LIN {X 0,Y 339.349,Z 929.895,A -85,B 0,C 180,E1 -14128.813,E2 -14128.813} C_VEL
LIN {X 0,Y 339.347,Z 930.371,A -85,B 0,C 180,E1 -14130,E2 -14130} C_VEL
LIN {X 0,Y 339.321,Z 930.387,A -85,B 0,C 180,E1 -14131.187,E2 -14131.187} C_VEL
LIN {X 0,Y 339.177,Z 929.963,A -85,B 0,C 180,E1 -14132.375,E2 -14132.375} C_VEL
LIN {X 0,Y 339.147,Z 929.133,A -85,B 0,C 180,E1 -14133.564,E2 -14133.564} C_VEL
LIN {X 0,Y 339.18,Z 927.893,A -85,B 0,C 180,E1 -14134.754,E2 -14134.754} C_VEL
LIN {X 0,Y 339.253,Z 925.189,A -85,B 0,C 180,E1 -14136.542,E2 -14136.542} C_VEL
LIN {X 0,Y 339.515,Z 921.472,A -85,B 0,C 180,E1 -14138.332,E2 -14138.332} C_VEL
LIN {X 0,Y 339.961,Z 916.67,A -85,B 0,C 180,E1 -14140.121,E2 -14140.121} C_VEL
LIN {X 0,Y 340.849,Z 909.521,A -85,B 0,C 180,E1 -14142.201,E2 -14142.201} C_VEL
LIN {X 0,Y 341.955,Z 901.959,A -85,B 0,C 180,E1 -14143.975,E2 -14143.975} C_VEL
LIN {X 0,Y 343.322,Z 892.798,A -85,B 0,C 180,E1 -14145.731,E2 -14145.731} C_VEL
LIN {X 0,Y 344.863,Z 882.415,A -85,B 0,C 180,E1 -14147.34,E2 -14147.34} C_VEL
LIN {X 0,Y 346.714,Z 871.123,A -85,B 0,C 180,E1 -14148.771,E2 -14148.771} C_VEL
LIN {X 0,Y 347.214,Z 865.96,A -85,B 0,C 180,E1 -14149.357,E2 -14149.357} C_VEL
LIN {X 0,Y 347.253,Z 853.333,A -85,B 0,C 180,E1 -14150.673,E2 -14150.673} C_VEL
LIN {X 0,Y 346.425,Z 843.606,A -85,B 0,C 180,E1 -14151.619,E2 -14151.619} C_VEL
LIN {X 0,Y 344.27,Z 832.038,A -85,B 0,C 180,E1 -14152.71,E2 -14152.71} C_VEL
LIN {X 0,Y 341.467,Z 821.968,A -85,B 0,C 180,E1 -14153.676,E2 -14153.676} C_VEL
LIN {X 0,Y 340.675,Z 818.661,A -85,B 0,C 180,E1 -14153.963,E2 -14153.963} C_VEL
LIN {X 0,Y 341.252,Z 813.344,A -85,B 0,C 180,E1 -14156.942,E2 -14156.942} C_VEL
LIN {X 0,Y 342.064,Z 807.69,A -85,B 0,C 180,E1 -14160.352,E2 -14160.352} C_VEL
LIN {X 0,Y 343.055,Z 802.834,A -85,B 0,C 180,E1 -14163.583,E2 -14163.583} C_VEL
LIN {X 0,Y 343.614,Z 799.164,A -85,B 0,C 180,E1 -14166.381,E2 -14166.381} C_VEL
LIN {X 0,Y 343.643,Z 796.286,A -85,B 0,C 180,E1 -14168.998,E2 -14168.998} C_VEL
LIN {X 0,Y 343.254,Z 793.267,A -85,B 0,C 180,E1 -14172.515,E2 -14172.515} C_VEL
LIN {X 0,Y 342.871,Z 791.214,A -85,B 0,C 180,E1 -14175.841,E2 -14175.841} C_VEL
LIN {X 0,Y 342.57,Z 789.841,A -85,B 0,C 180,E1 -14179.383,E2 -14179.383} C_VEL
LIN {X 0,Y 342.384,Z 789.323,A -85,B 0,C 180,E1 -14181.989,E2 -14181.989} C_VEL
LIN {X 0,Y 342.116,Z 789.226,A -85,B 0,C 180,E1 -14185.257,E2 -14185.257} C_VEL
LIN {X 0,Y 341.816,Z 789.514,A -85,B 0,C 180,E1 -14187.683,E2 -14187.683} C_VEL
LIN {X 0,Y 341.448,Z 790.146,A -85,B 0,C 180,E1 -14190.396,E2 -14190.396} C_VEL
LIN {X 0,Y 341.157,Z 791.012,A -85,B 0,C 180,E1 -14193.049,E2 -14193.049} C_VEL
LIN {X 0,Y 340.825,Z 792.487,A -85,B 0,C 180,E1 -14196.25,E2 -14196.25} C_VEL
LIN {X 0,Y 341.966,Z 795.393,A -85,B 0,C 180,E1 -14196.585,E2 -14196.585} C_VEL
LIN {X 0,Y 345.202,Z 802.217,A -85,B 0,C 180,E1 -14197.481,E2 -14197.481} C_VEL
LIN {X 0,Y 348.415,Z 810.639,A -85,B 0,C 180,E1 -14198.542,E2 -14198.542} C_VEL
LIN {X 0,Y 350.867,Z 820.747,A -85,B 0,C 180,E1 -14199.771,E2 -14199.771} C_VEL
LIN {X 0,Y 349.277,Z 832.605,A -85,B 0,C 180,E1 -14200.944,E2 -14200.944} C_VEL
LIN {X 0,Y 347.586,Z 843.821,A -85,B 0,C 180,E1 -14202.343,E2 -14202.343} C_VEL
LIN {X 0,Y 345.99,Z 853.23,A -85,B 0,C 180,E1 -14203.78,E2 -14203.78} C_VEL
LIN {X 0,Y 344.569,Z 861.071,A -85,B 0,C 180,E1 -14205.228,E2 -14205.228} C_VEL
LIN {X 0,Y 343.208,Z 868.826,A -85,B 0,C 180,E1 -14206.981,E2 -14206.981} C_VEL
LIN {X 0,Y 342.084,Z 875.111,A -85,B 0,C 180,E1 -14208.744,E2 -14208.744} C_VEL
LIN {X 0,Y 341.237,Z 880.125,A -85,B 0,C 180,E1 -14210.515,E2 -14210.515} C_VEL
LIN {X 0,Y 340.659,Z 883.491,A -85,B 0,C 180,E1 -14212.002,E2 -14212.002} C_VEL
LIN {X 0,Y 339.84,Z 886.98,A -85,B 0,C 180,E1 -14214.064,E2 -14214.064} C_VEL
LIN {X 0,Y 339.857,Z 888.363,A -85,B 0,C 180,E1 -14215.254,E2 -14215.254} C_VEL
LIN {X 0,Y 339.695,Z 889.321,A -85,B 0,C 180,E1 -14216.44,E2 -14216.44} C_VEL
LIN {X 0,Y 339.399,Z 890.044,A -85,B 0,C 180,E1 -14218.812,E2 -14218.812} C_VEL
LIN {X 0,Y 339.348,Z 889.81,A -85,B 0,C 180,E1 -14219.999,E2 -14219.999} C_VEL
LIN {X 0,Y 339.359,Z 889.126,A -85,B 0,C 180,E1 -14221.185,E2 -14221.185} C_VEL
LIN {X 0,Y 339.359,Z 888.038,A -85,B 0,C 180,E1 -14222.373,E2 -14222.373} C_VEL
LIN {X 0,Y 339.34,Z 886.549,A -85,B 0,C 180,E1 -14223.561,E2 -14223.561} C_VEL
LIN {X 0,Y 339.555,Z 883.457,A -85,B 0,C 180,E1 -14225.343,E2 -14225.343} C_VEL
LIN {X 0,Y 339.828,Z 879.306,A -85,B 0,C 180,E1 -14227.127,E2 -14227.127} C_VEL
LIN {X 0,Y 340.296,Z 872.949,A -85,B 0,C 180,E1 -14229.209,E2 -14229.209} C_VEL
LIN {X 0,Y 340.943,Z 866.043,A -85,B 0,C 180,E1 -14230.991,E2 -14230.991} C_VEL
LIN {X 0,Y 341.715,Z 857.519,A -85,B 0,C 180,E1 -14232.772,E2 -14232.772} C_VEL
LIN {X 0,Y 342.637,Z 848.818,A -85,B 0,C 180,E1 -14234.248,E2 -14234.248} C_VEL
LIN {X 0,Y 343.617,Z 838.67,A -85,B 0,C 180,E1 -14235.667,E2 -14235.667} C_VEL
LIN {X 0,Y 344.465,Z 827.918,A -85,B 0,C 180,E1 -14236.901,E2 -14236.901} C_VEL
LIN {X 0,Y 345.434,Z 815.586,A -85,B 0,C 180,E1 -14238.022,E2 -14238.022} C_VEL
LIN {X 0,Y 345.337,Z 812.445,A -85,B 0,C 180,E1 -14238.283,E2 -14238.283} C_VEL
LIN {X 0,Y 342.494,Z 799.34,A -85,B 0,C 180,E1 -14239.278,E2 -14239.278} C_VEL
LIN {X 0,Y 339.507,Z 785.356,A -85,B 0,C 180,E1 -14240.088,E2 -14240.088} C_VEL
LIN {X 0,Y 339.632,Z 781.305,A -85,B 0,C 180,E1 -14244.446,E2 -14244.446} C_VEL
LIN {X 0,Y 339.737,Z 779.169,A -85,B 0,C 180,E1 -14247.186,E2 -14247.186} C_VEL
LIN {X 0,Y 340.169,Z 779.109,A -85,B 0,C 180,E1 -14251.097,E2 -14251.097} C_VEL
LIN {X 0,Y 340.534,Z 779.069,A -85,B 0,C 180,E1 -14254.358,E2 -14254.358} C_VEL
LIN {X 0,Y 340.668,Z 779.051,A -85,B 0,C 180,E1 -14256.744,E2 -14256.744} C_VEL
LIN {X 0,Y 340.694,Z 779.044,A -85,B 0,C 180,E1 -14259.751,E2 -14259.751} C_VEL
LIN {X 0,Y 340.671,Z 779.05,A -85,B 0,C 180,E1 -14262.903,E2 -14262.903} C_VEL
LIN {X 0,Y 340.67,Z 779.05,A -85,B 0,C 180,E1 -14267.095,E2 -14267.095} C_VEL
LIN {X 0,Y 340.692,Z 779.044,A -85,B 0,C 180,E1 -14270.246,E2 -14270.246} C_VEL
LIN {X 0,Y 340.703,Z 779.043,A -85,B 0,C 180,E1 -14273.558,E2 -14273.558} C_VEL
LIN {X 0,Y 340.685,Z 779.044,A -85,B 0,C 180,E1 -14276.152,E2 -14276.152} C_VEL
LIN {X 0,Y 340.716,Z 779.041,A -85,B 0,C 180,E1 -14280.033,E2 -14280.033} C_VEL
LIN {X 0,Y 340.715,Z 779.044,A -85,B 0,C 180,E1 -14283.012,E2 -14283.012} C_VEL
LIN {X 0,Y 340.734,Z 779.041,A -85,B 0,C 180,E1 -14285.637,E2 -14285.637} C_VEL
LIN {X 0,Y 340.722,Z 779.046,A -85,B 0,C 180,E1 -14289.472,E2 -14289.472} C_VEL
LIN {X 0,Y 340.783,Z 779.034,A -85,B 0,C 180,E1 -14291.98,E2 -14291.98} C_VEL
LIN {X 0,Y 340.861,Z 779.028,A -85,B 0,C 180,E1 -14295.705,E2 -14295.705} C_VEL
LIN {X 0,Y 340.838,Z 779.028,A -85,B 0,C 180,E1 -14299.305,E2 -14299.305} C_VEL
LIN {X 0,Y 340.99,Z 779.006,A -85,B 0,C 180,E1 -14302.896,E2 -14302.896} C_VEL
LIN {X 0,Y 340.798,Z 779.031,A -85,B 0,C 180,E1 -14305.268,E2 -14305.268} C_VEL
LIN {X 0,Y 341.114,Z 778.994,A -85,B 0,C 180,E1 -14307.638,E2 -14307.638} C_VEL
LIN {X 0,Y 341.077,Z 778.995,A -85,B 0,C 180,E1 -14311.181,E2 -14311.181} C_VEL
LIN {X 0,Y 341.106,Z 778.995,A -85,B 0,C 180,E1 -14312.362,E2 -14312.362} C_VEL
LIN {X 0,Y 341.001,Z 779.008,A -85,B 0,C 180,E1 -14315.915,E2 -14315.915} C_VEL
LIN {X 0,Y 340.954,Z 779.016,A -85,B 0,C 180,E1 -14318.356,E2 -14318.356} C_VEL
LIN {X 0,Y 340.835,Z 779.028,A -85,B 0,C 180,E1 -14321.9,E2 -14321.9} C_VEL
LIN {X 0,Y 340.808,Z 779.029,A -85,B 0,C 180,E1 -14325.55,E2 -14325.55} C_VEL
LIN {X 0,Y 340.726,Z 779.039,A -85,B 0,C 180,E1 -14329.27,E2 -14329.27} C_VEL
LIN {X 0,Y 340.705,Z 779.044,A -85,B 0,C 180,E1 -14333.075,E2 -14333.075} C_VEL
LIN {X 0,Y 340.712,Z 779.041,A -85,B 0,C 180,E1 -14335.669,E2 -14335.669} C_VEL
LIN {X 0,Y 340.7,Z 779.043,A -85,B 0,C 180,E1 -14339.675,E2 -14339.675} C_VEL
LIN {X 0,Y 340.679,Z 779.047,A -85,B 0,C 180,E1 -14342.437,E2 -14342.437} C_VEL
LIN {X 0,Y 340.711,Z 779.044,A -85,B 0,C 180,E1 -14345.28,E2 -14345.28} C_VEL
LIN {X 0,Y 340.703,Z 779.043,A -85,B 0,C 180,E1 -14348.387,E2 -14348.387} C_VEL
LIN {X 0,Y 340.693,Z 779.044,A -85,B 0,C 180,E1 -14352.047,E2 -14352.047} C_VEL
LIN {X 0,Y 340.647,Z 779.049,A -85,B 0,C 180,E1 -14356.228,E2 -14356.228} C_VEL
LIN {X 0,Y 340.684,Z 779.047,A -85,B 0,C 180,E1 -14359.754,E2 -14359.754} C_VEL
LIN {X 0,Y 340.722,Z 779.043,A -85,B 0,C 180,E1 -14361.773,E2 -14361.773} C_VEL
LIN {X 0,Y 340.599,Z 779.055,A -85,B 0,C 180,E1 -14364.709,E2 -14364.709} C_VEL
LIN {X 0,Y 340.366,Z 779.088,A -85,B 0,C 180,E1 -14367.842,E2 -14367.842} C_VEL
LIN {X 0,Y 339.991,Z 779.131,A -85,B 0,C 180,E1 -14370.681,E2 -14370.681} C_VEL
LIN {X 0,Y 339.185,Z 779.237,A -85,B 0,C 180,E1 -14371.668,E2 -14371.668} C_VEL
LIN {X 0,Y 336.112,Z 779.617,A -85,B 0,C 180,E1 -14373.268,E2 -14373.268} C_VEL
LIN {X 0,Y 333.564,Z 780.155,A -85,B 0,C 180,E1 -14374.56,E2 -14374.56} C_VEL
LIN {X 0,Y 332.467,Z 780.857,A -85,B 0,C 180,E1 -14375.557,E2 -14375.557} C_VEL
LIN {X 0,Y 332.373,Z 781.177,A -85,B 0,C 180,E1 -14375.893,E2 -14375.893} C_VEL
LIN {X 0,Y 332.385,Z 785.144,A -85,B 0,C 180,E1 -14379.744,E2 -14379.744} C_VEL
LIN {X 0,Y 335.629,Z 800.339,A -85,B 0,C 180,E1 -14380.665,E2 -14380.665} C_VEL
LIN {X 0,Y 338.393,Z 814.066,A -85,B 0,C 180,E1 -14381.752,E2 -14381.752} C_VEL
LIN {X 0,Y 337.495,Z 826.677,A -85,B 0,C 180,E1 -14382.895,E2 -14382.895} C_VEL
LIN {X 0,Y 336.561,Z 838.501,A -85,B 0,C 180,E1 -14384.25,E2 -14384.25} C_VEL
LIN {X 0,Y 335.519,Z 849.022,A -85,B 0,C 180,E1 -14385.753,E2 -14385.753} C_VEL
LIN {X 0,Y 334.627,Z 857.724,A -85,B 0,C 180,E1 -14387.261,E2 -14387.261} C_VEL
LIN {X 0,Y 333.809,Z 866.28,A -85,B 0,C 180,E1 -14389.079,E2 -14389.079} C_VEL
LIN {X 0,Y 333.128,Z 873.174,A -85,B 0,C 180,E1 -14390.897,E2 -14390.897} C_VEL
LIN {X 0,Y 332.756,Z 878.716,A -85,B 0,C 180,E1 -14392.721,E2 -14392.721} C_VEL
LIN {X 0,Y 332.459,Z 883.055,A -85,B 0,C 180,E1 -14394.543,E2 -14394.543} C_VEL
LIN {X 0,Y 332.24,Z 886.294,A -85,B 0,C 180,E1 -14396.363,E2 -14396.363} C_VEL
LIN {X 0,Y 332.25,Z 887.903,A -85,B 0,C 180,E1 -14397.577,E2 -14397.577} C_VEL
LIN {X 0,Y 332.243,Z 889.056,A -85,B 0,C 180,E1 -14398.789,E2 -14398.789} C_VEL
LIN {X 0,Y 332.254,Z 889.818,A -85,B 0,C 180,E1 -14400.001,E2 -14400.001} C_VEL
LIN {X 0,Y 332.331,Z 890.18,A -85,B 0,C 180,E1 -14401.213,E2 -14401.213} C_VEL
LIN {X 0,Y 332.451,Z 890.086,A -85,B 0,C 180,E1 -14402.424,E2 -14402.424} C_VEL
LIN {X 0,Y 332.632,Z 889.594,A -85,B 0,C 180,E1 -14403.635,E2 -14403.635} C_VEL
LIN {X 0,Y 332.697,Z 888.725,A -85,B 0,C 180,E1 -14404.848,E2 -14404.848} C_VEL
LIN {X 0,Y 332.788,Z 887.425,A -85,B 0,C 180,E1 -14406.063,E2 -14406.063} C_VEL
LIN {X 0,Y 333.545,Z 884.458,A -85,B 0,C 180,E1 -14407.978,E2 -14407.978} C_VEL
LIN {X 0,Y 334.498,Z 879.384,A -85,B 0,C 180,E1 -14410.289,E2 -14410.289} C_VEL
LIN {X 0,Y 335.641,Z 873.077,A -85,B 0,C 180,E1 -14412.395,E2 -14412.395} C_VEL
LIN {X 0,Y 336.994,Z 866.267,A -85,B 0,C 180,E1 -14414.186,E2 -14414.186} C_VEL
LIN {X 0,Y 338.55,Z 857.938,A -85,B 0,C 180,E1 -14415.967,E2 -14415.967} C_VEL
LIN {X 0,Y 340.492,Z 847.529,A -85,B 0,C 180,E1 -14417.726,E2 -14417.726} C_VEL
LIN {X 0,Y 342.236,Z 836.91,A -85,B 0,C 180,E1 -14419.183,E2 -14419.183} C_VEL
LIN {X 0,Y 343.862,Z 826.568,A -85,B 0,C 180,E1 -14420.333,E2 -14420.333} C_VEL
LIN {X 0,Y 344.458,Z 822.579,A -85,B 0,C 180,E1 -14420.715,E2 -14420.715} C_VEL
LIN {X 0,Y 343.134,Z 815.08,A -85,B 0,C 180,E1 -14421.635,E2 -14421.635} C_VEL
LIN {X 0,Y 340.316,Z 806.149,A -85,B 0,C 180,E1 -14422.794,E2 -14422.794} C_VEL
LIN {X 0,Y 335.359,Z 794.765,A -85,B 0,C 180,E1 -14424.335,E2 -14424.335} C_VEL
LIN {X 0,Y 333.988,Z 791.924,A -85,B 0,C 180,E1 -14424.73,E2 -14424.73} C_VEL
LIN {X 0,Y 333.818,Z 791.217,A -85,B 0,C 180,E1 -14424.812,E2 -14424.812} C_VEL
LIN {X 0,Y 333.989,Z 788.694,A -85,B 0,C 180,E1 -14427.897,E2 -14427.897} C_VEL
LIN {X 0,Y 334.154,Z 786.738,A -85,B 0,C 180,E1 -14430.421,E2 -14430.421} C_VEL
LIN {X 0,Y 334.237,Z 784.77,A -85,B 0,C 180,E1 -14433.142,E2 -14433.142} C_VEL
LIN {X 0,Y 334.25,Z 783.55,A -85,B 0,C 180,E1 -14434.913,E2 -14434.913} C_VEL
LIN {X 0,Y 334.076,Z 782.019,A -85,B 0,C 180,E1 -14437.596,E2 -14437.596} C_VEL
LIN {X 0,Y 333.768,Z 780.568,A -85,B 0,C 180,E1 -14440.751,E2 -14440.751} C_VEL
LIN {X 0,Y 333.643,Z 779.925,A -85,B 0,C 180,E1 -14443.625,E2 -14443.625} C_VEL
LIN {X 0,Y 333.656,Z 780.06,A -85,B 0,C 180,E1 -14444.036,E2 -14444.036} C_VEL
LIN {X 0,Y 334.735,Z 785.742,A -85,B 0,C 180,E1 -14447.789,E2 -14447.789} C_VEL
LIN {X 0,Y 335.922,Z 792.316,A -85,B 0,C 180,E1 -14451.89,E2 -14451.89} C_VEL
LIN {X 0,Y 336.086,Z 796.175,A -85,B 0,C 180,E1 -14454.16,E2 -14454.16} C_VEL
LIN {X 0,Y 335.441,Z 801.211,A -85,B 0,C 180,E1 -14456.993,E2 -14456.993} C_VEL
LIN {X 0,Y 334.592,Z 807.453,A -85,B 0,C 180,E1 -14460.422,E2 -14460.422} C_VEL
LIN {X 0,Y 333.932,Z 813.667,A -85,B 0,C 180,E1 -14463.77,E2 -14463.77} C_VEL
LIN {X 0,Y 333.597,Z 816.798,A -85,B 0,C 180,E1 -14465.433,E2 -14465.433} C_VEL
LIN {X 0,Y 334.287,Z 820.354,A -85,B 0,C 180,E1 -14465.738,E2 -14465.738} C_VEL
LIN {X 0,Y 335.239,Z 823.541,A -85,B 0,C 180,E1 -14466.06,E2 -14466.06} C_VEL
LIN {X 0,Y 338.089,Z 835.619,A -85,B 0,C 180,E1 -14467.253,E2 -14467.253} C_VEL
LIN {X 0,Y 339.824,Z 848.508,A -85,B 0,C 180,E1 -14468.54,E2 -14468.54} C_VEL
LIN {X 0,Y 340.064,Z 861.381,A -85,B 0,C 180,E1 -14469.905,E2 -14469.905} C_VEL
LIN {X 0,Y 339.933,Z 869.253,A -85,B 0,C 180,E1 -14470.84,E2 -14470.84} C_VEL
LIN {X 0,Y 338.252,Z 879.576,A -85,B 0,C 180,E1 -14472.154,E2 -14472.154} C_VEL
LIN {X 0,Y 336.388,Z 891.075,A -85,B 0,C 180,E1 -14473.96,E2 -14473.96} C_VEL
LIN {X 0,Y 334.99,Z 900.109,A -85,B 0,C 180,E1 -14475.729,E2 -14475.729} C_VEL
LIN {X 0,Y 333.877,Z 907.662,A -85,B 0,C 180,E1 -14477.54,E2 -14477.54} C_VEL
LIN {X 0,Y 332.951,Z 914.779,A -85,B 0,C 180,E1 -14479.664,E2 -14479.664} C_VEL
LIN {X 0,Y 332.466,Z 919.546,A -85,B 0,C 180,E1 -14481.49,E2 -14481.49} C_VEL
LIN {X 0,Y 332.222,Z 923.218,A -85,B 0,C 180,E1 -14483.318,E2 -14483.318} C_VEL
LIN {X 0,Y 332.182,Z 925.886,A -85,B 0,C 180,E1 -14485.145,E2 -14485.145} C_VEL
LIN {X 0,Y 332.167,Z 928.401,A -85,B 0,C 180,E1 -14487.575,E2 -14487.575} C_VEL
LIN {X 0,Y 332.287,Z 929.342,A -85,B 0,C 180,E1 -14488.788,E2 -14488.788} C_VEL
LIN {X 0,Y 332.287,Z 929.855,A -85,B 0,C 180,E1 -14490,E2 -14490} C_VEL
LIN {X 0,Y 332.24,Z 929.94,A -85,B 0,C 180,E1 -14491.212,E2 -14491.212} C_VEL
LIN {X 0,Y 332.082,Z 929.552,A -85,B 0,C 180,E1 -14492.426,E2 -14492.426} C_VEL
LIN {X 0,Y 332.071,Z 928.763,A -85,B 0,C 180,E1 -14493.64,E2 -14493.64} C_VEL
LIN {X 0,Y 332.126,Z 926.087,A -85,B 0,C 180,E1 -14495.976,E2 -14495.976} C_VEL
LIN {X 0,Y 332.338,Z 922.651,A -85,B 0,C 180,E1 -14497.901,E2 -14497.901} C_VEL
LIN {X 0,Y 332.759,Z 918.308,A -85,B 0,C 180,E1 -14499.728,E2 -14499.728} C_VEL
LIN {X 0,Y 333.524,Z 911.814,A -85,B 0,C 180,E1 -14501.856,E2 -14501.856} C_VEL
LIN {X 0,Y 334.663,Z 904.863,A -85,B 0,C 180,E1 -14503.666,E2 -14503.666} C_VEL
LIN {X 0,Y 335.897,Z 896.416,A -85,B 0,C 180,E1 -14505.472,E2 -14505.472} C_VEL
LIN {X 0,Y 337.623,Z 886.149,A -85,B 0,C 180,E1 -14507.255,E2 -14507.255} C_VEL
LIN {X 0,Y 339.652,Z 874.643,A -85,B 0,C 180,E1 -14508.863,E2 -14508.863} C_VEL
LIN {X 0,Y 340.621,Z 867.209,A -85,B 0,C 180,E1 -14509.747,E2 -14509.747} C_VEL
LIN {X 0,Y 340.885,Z 854.388,A -85,B 0,C 180,E1 -14511.177,E2 -14511.177} C_VEL
LIN {X 0,Y 340.006,Z 843.877,A -85,B 0,C 180,E1 -14512.257,E2 -14512.257} C_VEL
LIN {X 0,Y 337.705,Z 831.851,A -85,B 0,C 180,E1 -14513.49,E2 -14513.49} C_VEL
LIN {X 0,Y 334.719,Z 821.415,A -85,B 0,C 180,E1 -14514.58,E2 -14514.58} C_VEL
LIN {X 0,Y 333.862,Z 817.819,A -85,B 0,C 180,E1 -14514.962,E2 -14514.962} C_VEL
LIN {X 0,Y 334.707,Z 811.23,A -85,B 0,C 180,E1 -14518.878,E2 -14518.878} C_VEL
LIN {X 0,Y 335.971,Z 804.707,A -85,B 0,C 180,E1 -14523.201,E2 -14523.201} C_VEL
LIN {X 0,Y 336.512,Z 801.322,A -85,B 0,C 180,E1 -14525.787,E2 -14525.787} C_VEL
LIN {X 0,Y 336.73,Z 799.309,A -85,B 0,C 180,E1 -14527.521,E2 -14527.521} C_VEL
LIN {X 0,Y 336.546,Z 796.558,A -85,B 0,C 180,E1 -14530.343,E2 -14530.343} C_VEL
LIN {X 0,Y 336.182,Z 794.07,A -85,B 0,C 180,E1 -14533.62,E2 -14533.62} C_VEL
LIN {X 0,Y 335.808,Z 792.216,A -85,B 0,C 180,E1 -14537.097,E2 -14537.097} C_VEL
LIN {X 0,Y 335.55,Z 791.062,A -85,B 0,C 180,E1 -14540.801,E2 -14540.801} C_VEL
LIN {X 0,Y 335.279,Z 790.71,A -85,B 0,C 180,E1 -14544.06,E2 -14544.06} C_VEL
LIN {X 0,Y 334.937,Z 790.88,A -85,B 0,C 180,E1 -14547.069,E2 -14547.069} C_VEL
LIN {X 0,Y 334.56,Z 791.372,A -85,B 0,C 180,E1 -14549.723,E2 -14549.723} C_VEL
LIN {X 0,Y 334.227,Z 792.16,A -85,B 0,C 180,E1 -14552.443,E2 -14552.443} C_VEL
LIN {X 0,Y 333.956,Z 793.392,A -85,B 0,C 180,E1 -14555.292,E2 -14555.292} C_VEL
LIN {X 0,Y 335.117,Z 796.322,A -85,B 0,C 180,E1 -14555.665,E2 -14555.665} C_VEL
LIN {X 0,Y 338.932,Z 804.012,A -85,B 0,C 180,E1 -14556.797,E2 -14556.797} C_VEL
LIN {X 0,Y 342.469,Z 813.543,A -85,B 0,C 180,E1 -14558.088,E2 -14558.088} C_VEL
LIN {X 0,Y 344.382,Z 821.286,A -85,B 0,C 180,E1 -14559.095,E2 -14559.095} C_VEL
LIN {X 0,Y 344.655,Z 823.065,A -85,B 0,C 180,E1 -14559.314,E2 -14559.314} C_VEL
LIN {X 0,Y 342.812,Z 834.991,A -85,B 0,C 180,E1 -14560.571,E2 -14560.571} C_VEL
LIN {X 0,Y 341.059,Z 845.785,A -85,B 0,C 180,E1 -14561.994,E2 -14561.994} C_VEL
LIN {X 0,Y 339.34,Z 854.919,A -85,B 0,C 180,E1 -14563.454,E2 -14563.454} C_VEL
LIN {X 0,Y 337.85,Z 862.531,A -85,B 0,C 180,E1 -14564.927,E2 -14564.927} C_VEL
LIN {X 0,Y 336.399,Z 870.054,A -85,B 0,C 180,E1 -14566.713,E2 -14566.713} C_VEL
LIN {X 0,Y 335.208,Z 876.212,A -85,B 0,C 180,E1 -14568.51,E2 -14568.51} C_VEL
LIN {X 0,Y 334.305,Z 881.115,A -85,B 0,C 180,E1 -14570.317,E2 -14570.317} C_VEL
LIN {X 0,Y 333.684,Z 884.383,A -85,B 0,C 180,E1 -14571.854,E2 -14571.854} C_VEL
LIN {X 0,Y 332.815,Z 887.705,A -85,B 0,C 180,E1 -14573.938,E2 -14573.938} C_VEL
LIN {X 0,Y 332.802,Z 889.018,A -85,B 0,C 180,E1 -14575.153,E2 -14575.153} C_VEL
LIN {X 0,Y 332.655,Z 889.91,A -85,B 0,C 180,E1 -14576.365,E2 -14576.365} C_VEL
LIN {X 0,Y 332.465,Z 890.419,A -85,B 0,C 180,E1 -14577.576,E2 -14577.576} C_VEL
LIN {X 0,Y 332.341,Z 890.536,A -85,B 0,C 180,E1 -14578.787,E2 -14578.787} C_VEL
LIN {X 0,Y 332.288,Z 890.214,A -85,B 0,C 180,E1 -14579.999,E2 -14579.999} C_VEL
LIN {X 0,Y 332.281,Z 889.474,A -85,B 0,C 180,E1 -14581.211,E2 -14581.211} C_VEL
LIN {X 0,Y 332.265,Z 888.341,A -85,B 0,C 180,E1 -14582.423,E2 -14582.423} C_VEL
LIN {X 0,Y 332.32,Z 885.829,A -85,B 0,C 180,E1 -14584.244,E2 -14584.244} C_VEL
LIN {X 0,Y 332.545,Z 882.302,A -85,B 0,C 180,E1 -14586.064,E2 -14586.064} C_VEL
LIN {X 0,Y 332.837,Z 877.664,A -85,B 0,C 180,E1 -14587.887,E2 -14587.887} C_VEL
LIN {X 0,Y 333.47,Z 870.676,A -85,B 0,C 180,E1 -14590.012,E2 -14590.012} C_VEL
LIN {X 0,Y 334.212,Z 863.104,A -85,B 0,C 180,E1 -14591.83,E2 -14591.83} C_VEL
LIN {X 0,Y 335.131,Z 853.762,A -85,B 0,C 180,E1 -14593.645,E2 -14593.645} C_VEL
LIN {X 0,Y 336.225,Z 843.113,A -85,B 0,C 180,E1 -14595.3,E2 -14595.3} C_VEL
LIN {X 0,Y 337.061,Z 833.492,A -85,B 0,C 180,E1 -14596.528,E2 -14596.528} C_VEL
LIN {X 0,Y 337.991,Z 822.236,A -85,B 0,C 180,E1 -14597.703,E2 -14597.703} C_VEL
LIN {X 0,Y 338.538,Z 814.552,A -85,B 0,C 180,E1 -14598.365,E2 -14598.365} C_VEL
LIN {X 0,Y 336.162,Z 803.156,A -85,B 0,C 180,E1 -14599.301,E2 -14599.301} C_VEL
LIN {X 0,Y 333.147,Z 789.188,A -85,B 0,C 180,E1 -14600.192,E2 -14600.192} C_VEL
LIN {X 0,Y 332.419,Z 785.706,A -85,B 0,C 180,E1 -14600.415,E2 -14600.415} C_VEL
LIN {X 0,Y 332.555,Z 781.777,A -85,B 0,C 180,E1 -14604.668,E2 -14604.668} C_VEL
LIN {X 0,Y 332.586,Z 780.276,A -85,B 0,C 180,E1 -14606.342,E2 -14606.342} C_VEL
LIN {X 0,Y 332.879,Z 780.017,A -85,B 0,C 180,E1 -14609.05,E2 -14609.05} C_VEL
LIN {X 0,Y 333.38,Z 779.954,A -85,B 0,C 180,E1 -14613.235,E2 -14613.235} C_VEL
LIN {X 0,Y 333.633,Z 779.926,A -85,B 0,C 180,E1 -14616.824,E2 -14616.824} C_VEL
LIN {X 0,Y 333.643,Z 779.928,A -85,B 0,C 180,E1 -14620.683,E2 -14620.683} C_VEL
LIN {X 0,Y 333.588,Z 779.93,A -85,B 0,C 180,E1 -14624.249,E2 -14624.249} C_VEL
LIN {X 0,Y 333.636,Z 779.923,A -85,B 0,C 180,E1 -14627.617,E2 -14627.617} C_VEL
LIN {X 0,Y 333.646,Z 779.925,A -85,B 0,C 180,E1 -14631.201,E2 -14631.201} C_VEL
LIN {X 0,Y 333.669,Z 779.918,A -85,B 0,C 180,E1 -14633.86,E2 -14633.86} C_VEL
LIN {X 0,Y 333.636,Z 779.925,A -85,B 0,C 180,E1 -14637.412,E2 -14637.412} C_VEL
LIN {X 0,Y 333.647,Z 779.925,A -85,B 0,C 180,E1 -14641.022,E2 -14641.022} C_VEL
LIN {X 0,Y 333.691,Z 779.919,A -85,B 0,C 180,E1 -14645.088,E2 -14645.088} C_VEL
LIN {X 0,Y 333.662,Z 779.921,A -85,B 0,C 180,E1 -14649.018,E2 -14649.018} C_VEL
LIN {X 0,Y 333.732,Z 779.916,A -85,B 0,C 180,E1 -14651.586,E2 -14651.586} C_VEL
LIN {X 0,Y 333.799,Z 779.908,A -85,B 0,C 180,E1 -14655.576,E2 -14655.576} C_VEL
LIN {X 0,Y 333.807,Z 779.902,A -85,B 0,C 180,E1 -14659.077,E2 -14659.077} C_VEL
LIN {X 0,Y 333.945,Z 779.884,A -85,B 0,C 180,E1 -14662.746,E2 -14662.746} C_VEL
LIN {X 0,Y 333.765,Z 779.907,A -85,B 0,C 180,E1 -14665.168,E2 -14665.168} C_VEL
LIN {X 0,Y 334.054,Z 779.873,A -85,B 0,C 180,E1 -14667.588,E2 -14667.588} C_VEL
LIN {X 0,Y 334.047,Z 779.871,A -85,B 0,C 180,E1 -14671.206,E2 -14671.206} C_VEL
LIN {X 0,Y 334.047,Z 779.874,A -85,B 0,C 180,E1 -14672.412,E2 -14672.412} C_VEL
LIN {X 0,Y 333.975,Z 779.885,A -85,B 0,C 180,E1 -14676.04,E2 -14676.04} C_VEL
LIN {X 0,Y 333.903,Z 779.893,A -85,B 0,C 180,E1 -14678.473,E2 -14678.473} C_VEL
LIN {X 0,Y 333.778,Z 779.909,A -85,B 0,C 180,E1 -14682.155,E2 -14682.155} C_VEL
LIN {X 0,Y 333.799,Z 779.906,A -85,B 0,C 180,E1 -14684.635,E2 -14684.635} C_VEL
LIN {X 0,Y 333.715,Z 779.918,A -85,B 0,C 180,E1 -14688.618,E2 -14688.618} C_VEL
LIN {X 0,Y 333.645,Z 779.924,A -85,B 0,C 180,E1 -14692.282,E2 -14692.282} C_VEL
LIN {X 0,Y 333.681,Z 779.919,A -85,B 0,C 180,E1 -14695.091,E2 -14695.091} C_VEL
LIN {X 0,Y 333.647,Z 779.925,A -85,B 0,C 180,E1 -14698.978,E2 -14698.978} C_VEL
LIN {X 0,Y 333.636,Z 779.925,A -85,B 0,C 180,E1 -14702.588,E2 -14702.588} C_VEL
LIN {X 0,Y 333.669,Z 779.918,A -85,B 0,C 180,E1 -14706.14,E2 -14706.14} C_VEL
LIN {X 0,Y 333.64,Z 779.927,A -85,B 0,C 180,E1 -14709.193,E2 -14709.193} C_VEL
LIN {X 0,Y 333.626,Z 779.924,A -85,B 0,C 180,E1 -14712.501,E2 -14712.501} C_VEL
LIN {X 0,Y 333.591,Z 779.929,A -85,B 0,C 180,E1 -14715.956,E2 -14715.956} C_VEL
LIN {X 0,Y 333.643,Z 779.927,A -85,B 0,C 180,E1 -14719.317,E2 -14719.317} C_VEL
LIN {X 0,Y 333.634,Z 779.926,A -85,B 0,C 180,E1 -14723.175,E2 -14723.175} C_VEL
LIN {X 0,Y 333.416,Z 779.95,A -85,B 0,C 180,E1 -14726.769,E2 -14726.769} C_VEL
LIN {X 0,Y 332.949,Z 780.008,A -85,B 0,C 180,E1 -14730.66,E2 -14730.66} C_VEL
LIN {X 0,Y 332.598,Z 780.057,A -85,B 0,C 180,E1 -14733.659,E2 -14733.659} C_VEL
LIN {X 0,Y 332.412,Z 780.25,A -85,B 0,C 180,E1 -14734.987,E2 -14734.987} C_VEL
LIN {X 0,Y 332.373,Z 781.177,A -85,B 0,C 180,E1 -14735.893,E2 -14735.893} C_VEL
LIN {X 0,Y 331.7,Z 781.923,A -85,B 0,C 180,E1 -14736.555,E2 -14736.555} C_VEL
LIN {X 0,Y 328.896,Z 783.25,A -85,B 0,C 180,E1 -14737.589,E2 -14737.589} C_VEL
LIN {X 0,Y 326.048,Z 784.591,A -85,B 0,C 180,E1 -14738.639,E2 -14738.639} C_VEL
LIN {X 0,Y 325.336,Z 785.358,A -85,B 0,C 180,E1 -14739.32,E2 -14739.32} C_VEL
LIN {X 0,Y 325.336,Z 785.56,A -85,B 0,C 180,E1 -14739.473,E2 -14739.473} C_VEL
LIN {X 0,Y 328.015,Z 798.231,A -85,B 0,C 180,E1 -14740.223,E2 -14740.223} C_VEL
LIN {X 0,Y 330.526,Z 810.559,A -85,B 0,C 180,E1 -14741.166,E2 -14741.166} C_VEL
LIN {X 0,Y 331.452,Z 815.622,A -85,B 0,C 180,E1 -14741.616,E2 -14741.616} C_VEL
LIN {X 0,Y 330.439,Z 828.22,A -85,B 0,C 180,E1 -14742.808,E2 -14742.808} C_VEL
LIN {X 0,Y 329.56,Z 838.861,A -85,B 0,C 180,E1 -14744.065,E2 -14744.065} C_VEL
LIN {X 0,Y 328.604,Z 848.44,A -85,B 0,C 180,E1 -14745.447,E2 -14745.447} C_VEL
LIN {X 0,Y 327.509,Z 858.906,A -85,B 0,C 180,E1 -14747.295,E2 -14747.295} C_VEL
LIN {X 0,Y 326.675,Z 867.273,A -85,B 0,C 180,E1 -14749.151,E2 -14749.151} C_VEL
LIN {X 0,Y 325.991,Z 874.059,A -85,B 0,C 180,E1 -14751.009,E2 -14751.009} C_VEL
LIN {X 0,Y 325.575,Z 880.352,A -85,B 0,C 180,E1 -14753.207,E2 -14753.207} C_VEL
LIN {X 0,Y 325.318,Z 884.356,A -85,B 0,C 180,E1 -14755.044,E2 -14755.044} C_VEL
LIN {X 0,Y 325.167,Z 886.467,A -85,B 0,C 180,E1 -14756.284,E2 -14756.284} C_VEL
LIN {X 0,Y 325.155,Z 888.161,A -85,B 0,C 180,E1 -14757.524,E2 -14757.524} C_VEL
LIN {X 0,Y 325.151,Z 889.387,A -85,B 0,C 180,E1 -14758.763,E2 -14758.763} C_VEL
LIN {X 0,Y 325.178,Z 890.199,A -85,B 0,C 180,E1 -14760.001,E2 -14760.001} C_VEL
LIN {X 0,Y 325.256,Z 890.618,A -85,B 0,C 180,E1 -14761.239,E2 -14761.239} C_VEL
LIN {X 0,Y 325.403,Z 890.61,A -85,B 0,C 180,E1 -14762.477,E2 -14762.477} C_VEL
LIN {X 0,Y 325.57,Z 890.174,A -85,B 0,C 180,E1 -14763.714,E2 -14763.714} C_VEL
LIN {X 0,Y 325.769,Z 888.167,A -85,B 0,C 180,E1 -14766.194,E2 -14766.194} C_VEL
LIN {X 0,Y 326.575,Z 885.339,A -85,B 0,C 180,E1 -14768.134,E2 -14768.134} C_VEL
LIN {X 0,Y 327.299,Z 881.83,A -85,B 0,C 180,E1 -14769.893,E2 -14769.893} C_VEL
LIN {X 0,Y 328.24,Z 877.099,A -85,B 0,C 180,E1 -14771.737,E2 -14771.737} C_VEL
LIN {X 0,Y 329.501,Z 871.141,A -85,B 0,C 180,E1 -14773.57,E2 -14773.57} C_VEL
LIN {X 0,Y 331.039,Z 863.777,A -85,B 0,C 180,E1 -14775.39,E2 -14775.39} C_VEL
LIN {X 0,Y 332.921,Z 854.764,A -85,B 0,C 180,E1 -14777.191,E2 -14777.191} C_VEL
LIN {X 0,Y 334.961,Z 843.79,A -85,B 0,C 180,E1 -14778.954,E2 -14778.954} C_VEL
LIN {X 0,Y 337.021,Z 832.226,A -85,B 0,C 180,E1 -14780.413,E2 -14780.413} C_VEL
LIN {X 0,Y 338.278,Z 823.752,A -85,B 0,C 180,E1 -14781.313,E2 -14781.313} C_VEL
LIN {X 0,Y 336.592,Z 815.478,A -85,B 0,C 180,E1 -14782.427,E2 -14782.427} C_VEL
LIN {X 0,Y 333.337,Z 805.903,A -85,B 0,C 180,E1 -14783.777,E2 -14783.777} C_VEL
LIN {X 0,Y 328.629,Z 795.665,A -85,B 0,C 180,E1 -14785.324,E2 -14785.324} C_VEL
LIN {X 0,Y 327.087,Z 792.658,A -85,B 0,C 180,E1 -14785.805,E2 -14785.805} C_VEL
LIN {X 0,Y 326.934,Z 791.983,A -85,B 0,C 180,E1 -14785.917,E2 -14785.917} C_VEL
LIN {X 0,Y 327.204,Z 789.152,A -85,B 0,C 180,E1 -14789.606,E2 -14789.606} C_VEL
LIN {X 0,Y 327.409,Z 786.666,A -85,B 0,C 180,E1 -14793.159,E2 -14793.159} C_VEL
LIN {X 0,Y 327.43,Z 785.298,A -85,B 0,C 180,E1 -14795.419,E2 -14795.419} C_VEL
LIN {X 0,Y 327.246,Z 783.734,A -85,B 0,C 180,E1 -14798.523,E2 -14798.523} C_VEL
LIN {X 0,Y 327.003,Z 782.644,A -85,B 0,C 180,E1 -14801.78,E2 -14801.78} C_VEL
LIN {X 0,Y 326.837,Z 782.201,A -85,B 0,C 180,E1 -14804.652,E2 -14804.652} C_VEL
LIN {X 0,Y 327.875,Z 787.731,A -85,B 0,C 180,E1 -14808.357,E2 -14808.357} C_VEL
LIN {X 0,Y 328.951,Z 793.852,A -85,B 0,C 180,E1 -14812.234,E2 -14812.234} C_VEL
LIN {X 0,Y 329.013,Z 797.251,A -85,B 0,C 180,E1 -14814.265,E2 -14814.265} C_VEL
LIN {X 0,Y 328.222,Z 803.125,A -85,B 0,C 180,E1 -14817.635,E2 -14817.635} C_VEL
LIN {X 0,Y 327.241,Z 810.585,A -85,B 0,C 180,E1 -14821.804,E2 -14821.804} C_VEL
LIN {X 0,Y 326.725,Z 815.293,A -85,B 0,C 180,E1 -14824.327,E2 -14824.327} C_VEL
LIN {X 0,Y 327.455,Z 818.877,A -85,B 0,C 180,E1 -14824.669,E2 -14824.669} C_VEL
LIN {X 0,Y 328.343,Z 821.577,A -85,B 0,C 180,E1 -14824.98,E2 -14824.98} C_VEL
LIN {X 0,Y 331.25,Z 833.228,A -85,B 0,C 180,E1 -14826.227,E2 -14826.227} C_VEL
LIN {X 0,Y 333.183,Z 845.898,A -85,B 0,C 180,E1 -14827.575,E2 -14827.575} C_VEL
LIN {X 0,Y 333.699,Z 855.121,A -85,B 0,C 180,E1 -14828.58,E2 -14828.58} C_VEL
LIN {X 0,Y 333.555,Z 868.155,A -85,B 0,C 180,E1 -14830.138,E2 -14830.138} C_VEL
LIN {X 0,Y 331.74,Z 879.484,A -85,B 0,C 180,E1 -14831.631,E2 -14831.631} C_VEL
LIN {X 0,Y 329.868,Z 890.187,A -85,B 0,C 180,E1 -14833.348,E2 -14833.348} C_VEL
LIN {X 0,Y 328.376,Z 899.088,A -85,B 0,C 180,E1 -14835.118,E2 -14835.118} C_VEL
LIN {X 0,Y 326.942,Z 907.874,A -85,B 0,C 180,E1 -14837.271,E2 -14837.271} C_VEL
LIN {X 0,Y 326.18,Z 912.971,A -85,B 0,C 180,E1 -14838.818,E2 -14838.818} C_VEL
LIN {X 0,Y 325.563,Z 917.995,A -85,B 0,C 180,E1 -14840.683,E2 -14840.683} C_VEL
LIN {X 0,Y 325.203,Z 921.929,A -85,B 0,C 180,E1 -14842.55,E2 -14842.55} C_VEL
LIN {X 0,Y 325.095,Z 924.222,A -85,B 0,C 180,E1 -14843.963,E2 -14843.963} C_VEL
LIN {X 0,Y 325.08,Z 925.574,A -85,B 0,C 180,E1 -14845.039,E2 -14845.039} C_VEL
LIN {X 0,Y 325.226,Z 928.774,A -85,B 0,C 180,E1 -14848.762,E2 -14848.762} C_VEL
LIN {X 0,Y 325.227,Z 929.326,A -85,B 0,C 180,E1 -14850,E2 -14850} C_VEL
LIN {X 0,Y 325.16,Z 929.458,A -85,B 0,C 180,E1 -14851.238,E2 -14851.238} C_VEL
LIN {X 0,Y 324.992,Z 929.147,A -85,B 0,C 180,E1 -14852.479,E2 -14852.479} C_VEL
LIN {X 0,Y 324.996,Z 928.4,A -85,B 0,C 180,E1 -14853.72,E2 -14853.72} C_VEL
LIN {X 0,Y 325.023,Z 926.06,A -85,B 0,C 180,E1 -14855.914,E2 -14855.914} C_VEL
LIN {X 0,Y 325.267,Z 922.473,A -85,B 0,C 180,E1 -14858.074,E2 -14858.074} C_VEL
LIN {X 0,Y 325.744,Z 918.25,A -85,B 0,C 180,E1 -14859.939,E2 -14859.939} C_VEL
LIN {X 0,Y 326.569,Z 911.908,A -85,B 0,C 180,E1 -14862.112,E2 -14862.112} C_VEL
LIN {X 0,Y 327.955,Z 903.855,A -85,B 0,C 180,E1 -14864.267,E2 -14864.267} C_VEL
LIN {X 0,Y 329.392,Z 895.388,A -85,B 0,C 180,E1 -14866.103,E2 -14866.103} C_VEL
LIN {X 0,Y 331.23,Z 884.996,A -85,B 0,C 180,E1 -14867.918,E2 -14867.918} C_VEL
LIN {X 0,Y 333.248,Z 874.634,A -85,B 0,C 180,E1 -14869.4,E2 -14869.4} C_VEL
LIN {X 0,Y 334.095,Z 868.698,A -85,B 0,C 180,E1 -14870.149,E2 -14870.149} C_VEL
LIN {X 0,Y 334.517,Z 855.349,A -85,B 0,C 180,E1 -14871.711,E2 -14871.711} C_VEL
LIN {X 0,Y 333.689,Z 844.397,A -85,B 0,C 180,E1 -14872.926,E2 -14872.926} C_VEL
LIN {X 0,Y 331.414,Z 832.574,A -85,B 0,C 180,E1 -14874.234,E2 -14874.234} C_VEL
LIN {X 0,Y 329.596,Z 825.629,A -85,B 0,C 180,E1 -14875.01,E2 -14875.01} C_VEL
LIN {X 0,Y 327.098,Z 817.753,A -85,B 0,C 180,E1 -14875.919,E2 -14875.919} C_VEL
LIN {X 0,Y 327.027,Z 816.966,A -85,B 0,C 180,E1 -14876.053,E2 -14876.053} C_VEL
LIN {X 0,Y 327.834,Z 811.373,A -85,B 0,C 180,E1 -14879.542,E2 -14879.542} C_VEL
LIN {X 0,Y 329.059,Z 805.523,A -85,B 0,C 180,E1 -14883.595,E2 -14883.595} C_VEL
LIN {X 0,Y 329.675,Z 801.738,A -85,B 0,C 180,E1 -14886.649,E2 -14886.649} C_VEL
LIN {X 0,Y 329.743,Z 800.098,A -85,B 0,C 180,E1 -14888.177,E2 -14888.177} C_VEL
LIN {X 0,Y 329.683,Z 798.483,A -85,B 0,C 180,E1 -14889.875,E2 -14889.875} C_VEL
LIN {X 0,Y 329.329,Z 796,A -85,B 0,C 180,E1 -14893.07,E2 -14893.07} C_VEL
LIN {X 0,Y 328.943,Z 794.023,A -85,B 0,C 180,E1 -14896.588,E2 -14896.588} C_VEL
LIN {X 0,Y 328.655,Z 792.784,A -85,B 0,C 180,E1 -14900.093,E2 -14900.093} C_VEL
LIN {X 0,Y 328.443,Z 792.274,A -85,B 0,C 180,E1 -14903.19,E2 -14903.19} C_VEL
LIN {X 0,Y 328.091,Z 792.275,A -85,B 0,C 180,E1 -14906.154,E2 -14906.154} C_VEL
LIN {X 0,Y 327.705,Z 792.671,A -85,B 0,C 180,E1 -14909.076,E2 -14909.076} C_VEL
LIN {X 0,Y 327.343,Z 793.343,A -85,B 0,C 180,E1 -14911.813,E2 -14911.813} C_VEL
LIN {X 0,Y 327.074,Z 794.175,A -85,B 0,C 180,E1 -14914.21,E2 -14914.21} C_VEL
LIN {X 0,Y 327.416,Z 795.474,A -85,B 0,C 180,E1 -14914.361,E2 -14914.361} C_VEL
LIN {X 0,Y 329.099,Z 798.226,A -85,B 0,C 180,E1 -14914.859,E2 -14914.859} C_VEL
LIN {X 0,Y 334.167,Z 809.457,A -85,B 0,C 180,E1 -14916.595,E2 -14916.595} C_VEL
LIN {X 0,Y 336.906,Z 817.553,A -85,B 0,C 180,E1 -14917.771,E2 -14917.771} C_VEL
LIN {X 0,Y 338.224,Z 823.372,A -85,B 0,C 180,E1 -14918.578,E2 -14918.578} C_VEL
LIN {X 0,Y 338.413,Z 825.344,A -85,B 0,C 180,E1 -14918.836,E2 -14918.836} C_VEL
LIN {X 0,Y 336.447,Z 837.241,A -85,B 0,C 180,E1 -14920.156,E2 -14920.156} C_VEL
LIN {X 0,Y 334.534,Z 847.853,A -85,B 0,C 180,E1 -14921.631,E2 -14921.631} C_VEL
LIN {X 0,Y 332.359,Z 858.248,A -85,B 0,C 180,E1 -14923.412,E2 -14923.412} C_VEL
LIN {X 0,Y 330.661,Z 866.645,A -85,B 0,C 180,E1 -14925.222,E2 -14925.222} C_VEL
LIN {X 0,Y 329.197,Z 873.505,A -85,B 0,C 180,E1 -14927.045,E2 -14927.045} C_VEL
LIN {X 0,Y 327.964,Z 879.036,A -85,B 0,C 180,E1 -14928.879,E2 -14928.879} C_VEL
LIN {X 0,Y 327.137,Z 883.409,A -85,B 0,C 180,E1 -14930.727,E2 -14930.727} C_VEL
LIN {X 0,Y 326.292,Z 886.766,A -85,B 0,C 180,E1 -14932.573,E2 -14932.573} C_VEL
LIN {X 0,Y 325.797,Z 888.472,A -85,B 0,C 180,E1 -14933.807,E2 -14933.807} C_VEL
LIN {X 0,Y 325.751,Z 889.678,A -85,B 0,C 180,E1 -14935.048,E2 -14935.048} C_VEL
LIN {X 0,Y 325.616,Z 890.506,A -85,B 0,C 180,E1 -14936.286,E2 -14936.286} C_VEL
LIN {X 0,Y 325.416,Z 890.959,A -85,B 0,C 180,E1 -14937.523,E2 -14937.523} C_VEL
LIN {X 0,Y 325.284,Z 891.006,A -85,B 0,C 180,E1 -14938.761,E2 -14938.761} C_VEL
LIN {X 0,Y 325.21,Z 890.611,A -85,B 0,C 180,E1 -14939.999,E2 -14939.999} C_VEL
LIN {X 0,Y 325.19,Z 889.818,A -85,B 0,C 180,E1 -14941.237,E2 -14941.237} C_VEL
LIN {X 0,Y 325.172,Z 888.629,A -85,B 0,C 180,E1 -14942.476,E2 -14942.476} C_VEL
LIN {X 0,Y 325.258,Z 886.009,A -85,B 0,C 180,E1 -14944.336,E2 -14944.336} C_VEL
LIN {X 0,Y 325.475,Z 882.373,A -85,B 0,C 180,E1 -14946.197,E2 -14946.197} C_VEL
LIN {X 0,Y 325.778,Z 877.628,A -85,B 0,C 180,E1 -14948.059,E2 -14948.059} C_VEL
LIN {X 0,Y 326.464,Z 870.48,A -85,B 0,C 180,E1 -14950.229,E2 -14950.229} C_VEL
LIN {X 0,Y 327.206,Z 862.797,A -85,B 0,C 180,E1 -14952.087,E2 -14952.087} C_VEL
LIN {X 0,Y 327.996,Z 855.013,A -85,B 0,C 180,E1 -14953.631,E2 -14953.631} C_VEL
LIN {X 0,Y 329.098,Z 844.55,A -85,B 0,C 180,E1 -14955.322,E2 -14955.322} C_VEL
LIN {X 0,Y 330.112,Z 833.651,A -85,B 0,C 180,E1 -14956.755,E2 -14956.755} C_VEL
LIN {X 0,Y 331.021,Z 822.605,A -85,B 0,C 180,E1 -14957.928,E2 -14957.928} C_VEL
LIN {X 0,Y 331.583,Z 815.731,A -85,B 0,C 180,E1 -14958.536,E2 -14958.536} C_VEL
LIN {X 0,Y 329.101,Z 803.705,A -85,B 0,C 180,E1 -14959.558,E2 -14959.558} C_VEL
LIN {X 0,Y 326.256,Z 790.418,A -85,B 0,C 180,E1 -14960.441,E2 -14960.441} C_VEL
LIN {X 0,Y 325.359,Z 786.076,A -85,B 0,C 180,E1 -14960.713,E2 -14960.713} C_VEL
LIN {X 0,Y 325.508,Z 782.228,A -85,B 0,C 180,E1 -14964.93,E2 -14964.93} C_VEL
LIN {X 0,Y 325.587,Z 780.931,A -85,B 0,C 180,E1 -14966.954,E2 -14966.954} C_VEL
LIN {X 0,Y 326.054,Z 780.867,A -85,B 0,C 180,E1 -14971.15,E2 -14971.15} C_VEL
LIN {X 0,Y 326.381,Z 780.828,A -85,B 0,C 180,E1 -14974.044,E2 -14974.044} C_VEL
LIN {X 0,Y 326.602,Z 780.799,A -85,B 0,C 180,E1 -14977.232,E2 -14977.232} C_VEL
LIN {X 0,Y 326.586,Z 780.803,A -85,B 0,C 180,E1 -14980.208,E2 -14980.208} C_VEL
LIN {X 0,Y 326.557,Z 780.804,A -85,B 0,C 180,E1 -14983.524,E2 -14983.524} C_VEL
LIN {X 0,Y 326.57,Z 780.806,A -85,B 0,C 180,E1 -14987.027,E2 -14987.027} C_VEL
LIN {X 0,Y 326.605,Z 780.803,A -85,B 0,C 180,E1 -14990.772,E2 -14990.772} C_VEL
LIN {X 0,Y 326.605,Z 780.799,A -85,B 0,C 180,E1 -14994.479,E2 -14994.479} C_VEL
LIN {X 0,Y 326.6,Z 780.801,A -85,B 0,C 180,E1 -14997.455,E2 -14997.455} C_VEL
LIN {X 0,Y 326.609,Z 780.798,A -85,B 0,C 180,E1 -15000.336,E2 -15000.336} C_VEL
LIN {X 0,Y 326.635,Z 780.795,A -85,B 0,C 180,E1 -15004.643,E2 -15004.643} C_VEL
LIN {X 0,Y 326.609,Z 780.798,A -85,B 0,C 180,E1 -15008.543,E2 -15008.543} C_VEL
LIN {X 0,Y 326.655,Z 780.792,A -85,B 0,C 180,E1 -15012.47,E2 -15012.47} C_VEL
LIN {X 0,Y 326.75,Z 780.78,A -85,B 0,C 180,E1 -15016.314,E2 -15016.314} C_VEL
LIN {X 0,Y 326.773,Z 780.78,A -85,B 0,C 180,E1 -15020.092,E2 -15020.092} C_VEL
LIN {X 0,Y 326.93,Z 780.764,A -85,B 0,C 180,E1 -15023.83,E2 -15023.83} C_VEL
LIN {X 0,Y 326.997,Z 780.751,A -85,B 0,C 180,E1 -15027.536,E2 -15027.536} C_VEL
LIN {X 0,Y 327.017,Z 780.747,A -85,B 0,C 180,E1 -15031.231,E2 -15031.231} C_VEL
LIN {X 0,Y 326.725,Z 780.785,A -85,B 0,C 180,E1 -15033.7,E2 -15033.7} C_VEL
LIN {X 0,Y 326.929,Z 780.764,A -85,B 0,C 180,E1 -15036.17,E2 -15036.17} C_VEL
LIN {X 0,Y 326.771,Z 780.78,A -85,B 0,C 180,E1 -15039.908,E2 -15039.908} C_VEL
LIN {X 0,Y 326.749,Z 780.781,A -85,B 0,C 180,E1 -15043.686,E2 -15043.686} C_VEL
LIN {X 0,Y 326.655,Z 780.792,A -85,B 0,C 180,E1 -15047.53,E2 -15047.53} C_VEL
LIN {X 0,Y 326.609,Z 780.797,A -85,B 0,C 180,E1 -15051.457,E2 -15051.457} C_VEL
LIN {X 0,Y 326.627,Z 780.796,A -85,B 0,C 180,E1 -15055.489,E2 -15055.489} C_VEL
LIN {X 0,Y 326.609,Z 780.798,A -85,B 0,C 180,E1 -15059.664,E2 -15059.664} C_VEL
LIN {X 0,Y 326.61,Z 780.803,A -85,B 0,C 180,E1 -15062.947,E2 -15062.947} C_VEL
LIN {X 0,Y 326.605,Z 780.799,A -85,B 0,C 180,E1 -15065.521,E2 -15065.521} C_VEL
LIN {X 0,Y 326.605,Z 780.803,A -85,B 0,C 180,E1 -15069.228,E2 -15069.228} C_VEL
LIN {X 0,Y 326.57,Z 780.806,A -85,B 0,C 180,E1 -15072.973,E2 -15072.973} C_VEL
LIN {X 0,Y 326.571,Z 780.806,A -85,B 0,C 180,E1 -15077.029,E2 -15077.029} C_VEL
LIN {X 0,Y 326.605,Z 780.799,A -85,B 0,C 180,E1 -15080.775,E2 -15080.775} C_VEL
LIN {X 0,Y 326.605,Z 780.8,A -85,B 0,C 180,E1 -15082.952,E2 -15082.952} C_VEL
LIN {X 0,Y 326.419,Z 780.824,A -85,B 0,C 180,E1 -15085.96,E2 -15085.96} C_VEL
LIN {X 0,Y 326.105,Z 780.861,A -85,B 0,C 180,E1 -15088.855,E2 -15088.855} C_VEL
LIN {X 0,Y 325.73,Z 780.909,A -85,B 0,C 180,E1 -15092.206,E2 -15092.206} C_VEL
LIN {X 0,Y 325.352,Z 781.081,A -85,B 0,C 180,E1 -15095.129,E2 -15095.129} C_VEL
LIN {X 0,Y 325.336,Z 785.358,A -85,B 0,C 180,E1 -15099.32,E2 -15099.32} C_VEL
LIN {X 0,Y 325.32,Z 786.457,A -85,B 0,C 180,E1 -15099.504,E2 -15099.504} C_VEL
LIN {X 0,Y 325.236,Z 799.788,A -85,B 0,C 180,E1 -15100.2,E2 -15100.2} C_VEL
LIN {X 0,Y 324.637,Z 805.178,A -85,B 0,C 180,E1 -15100.533,E2 -15100.533} C_VEL
LIN {X 0,Y 324.01,Z 811.104,A -85,B 0,C 180,E1 -15100.909,E2 -15100.909} C_VEL
LIN {X 0,Y 324.211,Z 814.859,A -85,B 0,C 180,E1 -15101.274,E2 -15101.274} C_VEL
LIN {X 0,Y 324.239,Z 819.385,A -85,B 0,C 180,E1 -15101.683,E2 -15101.683} C_VEL
LIN {X 0,Y 323.317,Z 830.231,A -85,B 0,C 180,E1 -15102.784,E2 -15102.784} C_VEL
LIN {X 0,Y 322.215,Z 842.451,A -85,B 0,C 180,E1 -15104.342,E2 -15104.342} C_VEL
LIN {X 0,Y 321.258,Z 851.514,A -85,B 0,C 180,E1 -15105.754,E2 -15105.754} C_VEL
LIN {X 0,Y 320.23,Z 861.397,A -85,B 0,C 180,E1 -15107.646,E2 -15107.646} C_VEL
LIN {X 0,Y 319.432,Z 869.432,A -85,B 0,C 180,E1 -15109.544,E2 -15109.544} C_VEL
LIN {X 0,Y 318.866,Z 874.903,A -85,B 0,C 180,E1 -15111.126,E2 -15111.126} C_VEL
LIN {X 0,Y 318.467,Z 880.812,A -85,B 0,C 180,E1 -15113.252,E2 -15113.252} C_VEL
LIN {X 0,Y 318.18,Z 885.609,A -85,B 0,C 180,E1 -15115.567,E2 -15115.567} C_VEL
LIN {X 0,Y 318.061,Z 888.39,A -85,B 0,C 180,E1 -15117.468,E2 -15117.468} C_VEL
LIN {X 0,Y 318.059,Z 889.711,A -85,B 0,C 180,E1 -15118.735,E2 -15118.735} C_VEL
LIN {X 0,Y 318.088,Z 890.577,A -85,B 0,C 180,E1 -15120.001,E2 -15120.001} C_VEL
LIN {X 0,Y 318.184,Z 891.048,A -85,B 0,C 180,E1 -15121.267,E2 -15121.267} C_VEL
LIN {X 0,Y 318.337,Z 891.129,A -85,B 0,C 180,E1 -15122.532,E2 -15122.532} C_VEL
LIN {X 0,Y 318.51,Z 890.772,A -85,B 0,C 180,E1 -15123.797,E2 -15123.797} C_VEL
LIN {X 0,Y 318.753,Z 888.873,A -85,B 0,C 180,E1 -15126.331,E2 -15126.331} C_VEL
LIN {X 0,Y 319.596,Z 886.219,A -85,B 0,C 180,E1 -15128.284,E2 -15128.284} C_VEL
LIN {X 0,Y 320.376,Z 882.81,A -85,B 0,C 180,E1 -15130.109,E2 -15130.109} C_VEL
LIN {X 0,Y 321.38,Z 878.231,A -85,B 0,C 180,E1 -15131.992,E2 -15131.992} C_VEL
LIN {X 0,Y 323.014,Z 871.324,A -85,B 0,C 180,E1 -15134.17,E2 -15134.17} C_VEL
LIN {X 0,Y 324.688,Z 863.993,A -85,B 0,C 180,E1 -15136.022,E2 -15136.022} C_VEL
LIN {X 0,Y 326.7,Z 854.949,A -85,B 0,C 180,E1 -15137.852,E2 -15137.852} C_VEL
LIN {X 0,Y 328.881,Z 844.124,A -85,B 0,C 180,E1 -15139.617,E2 -15139.617} C_VEL
LIN {X 0,Y 330.935,Z 833.501,A -85,B 0,C 180,E1 -15141.001,E2 -15141.001} C_VEL
LIN {X 0,Y 332.223,Z 825.94,A -85,B 0,C 180,E1 -15141.836,E2 -15141.836} C_VEL
LIN {X 0,Y 330.543,Z 817.604,A -85,B 0,C 180,E1 -15143.034,E2 -15143.034} C_VEL
LIN {X 0,Y 326.878,Z 806.949,A -85,B 0,C 180,E1 -15144.668,E2 -15144.668} C_VEL
LIN {X 0,Y 321.981,Z 796.701,A -85,B 0,C 180,E1 -15146.406,E2 -15146.406} C_VEL
LIN {X 0,Y 320.337,Z 793.611,A -85,B 0,C 180,E1 -15146.972,E2 -15146.972} C_VEL
LIN {X 0,Y 320.124,Z 792.838,A -85,B 0,C 180,E1 -15147.088,E2 -15147.088} C_VEL
LIN {X 0,Y 320.397,Z 790.525,A -85,B 0,C 180,E1 -15150.3,E2 -15150.3} C_VEL
LIN {X 0,Y 320.617,Z 788.404,A -85,B 0,C 180,E1 -15153.595,E2 -15153.595} C_VEL
LIN {X 0,Y 320.617,Z 786.971,A -85,B 0,C 180,E1 -15156.289,E2 -15156.289} C_VEL
LIN {X 0,Y 320.448,Z 785.554,A -85,B 0,C 180,E1 -15159.86,E2 -15159.86} C_VEL
LIN {X 0,Y 320.33,Z 784.824,A -85,B 0,C 180,E1 -15163.613,E2 -15163.613} C_VEL
LIN {X 0,Y 320.179,Z 785.026,A -85,B 0,C 180,E1 -15165.805,E2 -15165.805} C_VEL
LIN {X 0,Y 321.017,Z 789.695,A -85,B 0,C 180,E1 -15168.944,E2 -15168.944} C_VEL
LIN {X 0,Y 321.919,Z 794.918,A -85,B 0,C 180,E1 -15172.317,E2 -15172.317} C_VEL
LIN {X 0,Y 321.986,Z 797.483,A -85,B 0,C 180,E1 -15173.89,E2 -15173.89} C_VEL
LIN {X 0,Y 321.337,Z 802.507,A -85,B 0,C 180,E1 -15176.854,E2 -15176.854} C_VEL
LIN {X 0,Y 320.453,Z 808.724,A -85,B 0,C 180,E1 -15180.432,E2 -15180.432} C_VEL
LIN {X 0,Y 319.926,Z 813.345,A -85,B 0,C 180,E1 -15183.059,E2 -15183.059} C_VEL
LIN {X 0,Y 320.585,Z 817.024,A -85,B 0,C 180,E1 -15183.433,E2 -15183.433} C_VEL
LIN {X 0,Y 321.571,Z 819.717,A -85,B 0,C 180,E1 -15183.797,E2 -15183.797} C_VEL
LIN {X 0,Y 324.833,Z 832.88,A -85,B 0,C 180,E1 -15185.329,E2 -15185.329} C_VEL
LIN {X 0,Y 326.81,Z 845.126,A -85,B 0,C 180,E1 -15186.737,E2 -15186.737} C_VEL
LIN {X 0,Y 327.436,Z 856.229,A -85,B 0,C 180,E1 -15188.024,E2 -15188.024} C_VEL
LIN {X 0,Y 327.049,Z 868.481,A -85,B 0,C 180,E1 -15189.562,E2 -15189.562} C_VEL
LIN {X 0,Y 326.518,Z 873.148,A -85,B 0,C 180,E1 -15190.184,E2 -15190.184} C_VEL
LIN {X 0,Y 324.548,Z 883.478,A -85,B 0,C 180,E1 -15191.7,E2 -15191.7} C_VEL
LIN {X 0,Y 322.575,Z 893.751,A -85,B 0,C 180,E1 -15193.547,E2 -15193.547} C_VEL
LIN {X 0,Y 321.016,Z 902.192,A -85,B 0,C 180,E1 -15195.418,E2 -15195.418} C_VEL
LIN {X 0,Y 319.614,Z 910.174,A -85,B 0,C 180,E1 -15197.62,E2 -15197.62} C_VEL
LIN {X 0,Y 318.721,Z 916.451,A -85,B 0,C 180,E1 -15199.84,E2 -15199.84} C_VEL
LIN {X 0,Y 318.228,Z 920.614,A -85,B 0,C 180,E1 -15201.747,E2 -15201.747} C_VEL
LIN {X 0,Y 317.996,Z 924.218,A -85,B 0,C 180,E1 -15204.019,E2 -15204.019} C_VEL
LIN {X 0,Y 317.948,Z 926.4,A -85,B 0,C 180,E1 -15206.198,E2 -15206.198} C_VEL
LIN {X 0,Y 318.165,Z 928.196,A -85,B 0,C 180,E1 -15208.734,E2 -15208.734} C_VEL
LIN {X 0,Y 318.169,Z 928.793,A -85,B 0,C 180,E1 -15210,E2 -15210} C_VEL
LIN {X 0,Y 318.081,Z 928.967,A -85,B 0,C 180,E1 -15211.266,E2 -15211.266} C_VEL
LIN {X 0,Y 317.904,Z 928.722,A -85,B 0,C 180,E1 -15212.534,E2 -15212.534} C_VEL
LIN {X 0,Y 317.922,Z 928.039,A -85,B 0,C 180,E1 -15213.803,E2 -15213.803} C_VEL
LIN {X 0,Y 317.972,Z 925.412,A -85,B 0,C 180,E1 -15216.345,E2 -15216.345} C_VEL
LIN {X 0,Y 318.214,Z 922.315,A -85,B 0,C 180,E1 -15218.254,E2 -15218.254} C_VEL
LIN {X 0,Y 318.721,Z 918.189,A -85,B 0,C 180,E1 -15220.16,E2 -15220.16} C_VEL
LIN {X 0,Y 319.443,Z 913.01,A -85,B 0,C 180,E1 -15222.064,E2 -15222.064} C_VEL
LIN {X 0,Y 320.888,Z 905.445,A -85,B 0,C 180,E1 -15224.264,E2 -15224.264} C_VEL
LIN {X 0,Y 322.602,Z 895.904,A -85,B 0,C 180,E1 -15226.452,E2 -15226.452} C_VEL
LIN {X 0,Y 324.541,Z 885.932,A -85,B 0,C 180,E1 -15228.301,E2 -15228.301} C_VEL
LIN {X 0,Y 326.862,Z 874.737,A -85,B 0,C 180,E1 -15229.958,E2 -15229.958} C_VEL
LIN {X 0,Y 327.654,Z 868.96,A -85,B 0,C 180,E1 -15230.727,E2 -15230.727} C_VEL
LIN {X 0,Y 328.239,Z 856.452,A -85,B 0,C 180,E1 -15232.275,E2 -15232.275} C_VEL
LIN {X 0,Y 327.475,Z 845.516,A -85,B 0,C 180,E1 -15233.561,E2 -15233.561} C_VEL
LIN {X 0,Y 325.248,Z 833.346,A -85,B 0,C 180,E1 -15235.015,E2 -15235.015} C_VEL
LIN {X 0,Y 321.953,Z 821.555,A -85,B 0,C 180,E1 -15236.49,E2 -15236.49} C_VEL
LIN {X 0,Y 320.403,Z 817.4,A -85,B 0,C 180,E1 -15237.05,E2 -15237.05} C_VEL
LIN {X 0,Y 320.24,Z 816.176,A -85,B 0,C 180,E1 -15237.204,E2 -15237.204} C_VEL
LIN {X 0,Y 320.992,Z 811.557,A -85,B 0,C 180,E1 -15240.237,E2 -15240.237} C_VEL
LIN {X 0,Y 322.16,Z 806.357,A -85,B 0,C 180,E1 -15244.004,E2 -15244.004} C_VEL
LIN {X 0,Y 322.667,Z 803.577,A -85,B 0,C 180,E1 -15246.302,E2 -15246.302} C_VEL
LIN {X 0,Y 322.737,Z 800.66,A -85,B 0,C 180,E1 -15249.162,E2 -15249.162} C_VEL
LIN {X 0,Y 322.482,Z 798.187,A -85,B 0,C 180,E1 -15252.184,E2 -15252.184} C_VEL
LIN {X 0,Y 322.118,Z 796.018,A -85,B 0,C 180,E1 -15255.718,E2 -15255.718} C_VEL
LIN {X 0,Y 321.759,Z 794.427,A -85,B 0,C 180,E1 -15259.861,E2 -15259.861} C_VEL
LIN {X 0,Y 321.594,Z 793.929,A -85,B 0,C 180,E1 -15262.272,E2 -15262.272} C_VEL
LIN {X 0,Y 321.254,Z 793.745,A -85,B 0,C 180,E1 -15265.332,E2 -15265.332} C_VEL
LIN {X 0,Y 320.796,Z 794.067,A -85,B 0,C 180,E1 -15268.695,E2 -15268.695} C_VEL
LIN {X 0,Y 320.209,Z 795.103,A -85,B 0,C 180,E1 -15272.99,E2 -15272.99} C_VEL
LIN {X 0,Y 320.726,Z 796.777,A -85,B 0,C 180,E1 -15273.235,E2 -15273.235} C_VEL
LIN {X 0,Y 324.56,Z 803.562,A -85,B 0,C 180,E1 -15274.533,E2 -15274.533} C_VEL
LIN {X 0,Y 329.068,Z 814.181,A -85,B 0,C 180,E1 -15276.305,E2 -15276.305} C_VEL
LIN {X 0,Y 331.671,Z 823.18,A -85,B 0,C 180,E1 -15277.698,E2 -15277.698} C_VEL
LIN {X 0,Y 332.246,Z 827.741,A -85,B 0,C 180,E1 -15278.332,E2 -15278.332} C_VEL
LIN {X 0,Y 330.294,Z 838.679,A -85,B 0,C 180,E1 -15279.608,E2 -15279.608} C_VEL
LIN {X 0,Y 328.03,Z 849.929,A -85,B 0,C 180,E1 -15281.253,E2 -15281.253} C_VEL
LIN {X 0,Y 326.132,Z 858.489,A -85,B 0,C 180,E1 -15282.763,E2 -15282.763} C_VEL
LIN {X 0,Y 324.492,Z 865.634,A -85,B 0,C 180,E1 -15284.291,E2 -15284.291} C_VEL
LIN {X 0,Y 322.874,Z 872.713,A -85,B 0,C 180,E1 -15286.145,E2 -15286.145} C_VEL
LIN {X 0,Y 321.526,Z 878.496,A -85,B 0,C 180,E1 -15288.014,E2 -15288.014} C_VEL
LIN {X 0,Y 320.454,Z 883.091,A -85,B 0,C 180,E1 -15289.894,E2 -15289.894} C_VEL
LIN {X 0,Y 319.775,Z 886.169,A -85,B 0,C 180,E1 -15291.499,E2 -15291.499} C_VEL
LIN {X 0,Y 318.779,Z 889.201,A -85,B 0,C 180,E1 -15293.67,E2 -15293.67} C_VEL
LIN {X 0,Y 318.706,Z 890.349,A -85,B 0,C 180,E1 -15294.938,E2 -15294.938} C_VEL
LIN {X 0,Y 318.578,Z 891.12,A -85,B 0,C 180,E1 -15296.204,E2 -15296.204} C_VEL
LIN {X 0,Y 318.369,Z 891.508,A -85,B 0,C 180,E1 -15297.468,E2 -15297.468} C_VEL
LIN {X 0,Y 318.21,Z 891.455,A -85,B 0,C 180,E1 -15298.733,E2 -15298.733} C_VEL
LIN {X 0,Y 318.135,Z 891.001,A -85,B 0,C 180,E1 -15299.999,E2 -15299.999} C_VEL
LIN {X 0,Y 318.098,Z 890.155,A -85,B 0,C 180,E1 -15301.265,E2 -15301.265} C_VEL
LIN {X 0,Y 318.078,Z 888.894,A -85,B 0,C 180,E1 -15302.531,E2 -15302.531} C_VEL
LIN {X 0,Y 318.196,Z 886.172,A -85,B 0,C 180,E1 -15304.432,E2 -15304.432} C_VEL
LIN {X 0,Y 318.474,Z 881.409,A -85,B 0,C 180,E1 -15306.758,E2 -15306.758} C_VEL
LIN {X 0,Y 318.876,Z 875.628,A -85,B 0,C 180,E1 -15308.874,E2 -15308.874} C_VEL
LIN {X 0,Y 319.54,Z 869.034,A -85,B 0,C 180,E1 -15310.773,E2 -15310.773} C_VEL
LIN {X 0,Y 320.346,Z 860.85,A -85,B 0,C 180,E1 -15312.672,E2 -15312.672} C_VEL
LIN {X 0,Y 321.485,Z 850.786,A -85,B 0,C 180,E1 -15314.559,E2 -15314.559} C_VEL
LIN {X 0,Y 322.578,Z 840.383,A -85,B 0,C 180,E1 -15316.127,E2 -15316.127} C_VEL
LIN {X 0,Y 323.543,Z 828.974,A -85,B 0,C 180,E1 -15317.532,E2 -15317.532} C_VEL
LIN {X 0,Y 324.524,Z 817.835,A -85,B 0,C 180,E1 -15318.627,E2 -15318.627} C_VEL
LIN {X 0,Y 324.091,Z 814.013,A -85,B 0,C 180,E1 -15318.981,E2 -15318.981} C_VEL
LIN {X 0,Y 321.324,Z 800.802,A -85,B 0,C 180,E1 -15320.061,E2 -15320.061} C_VEL
LIN {X 0,Y 318.379,Z 787.054,A -85,B 0,C 180,E1 -15320.93,E2 -15320.93} C_VEL
LIN {X 0,Y 318.333,Z 786.502,A -85,B 0,C 180,E1 -15320.959,E2 -15320.959} C_VEL
LIN {X 0,Y 318.443,Z 782.692,A -85,B 0,C 180,E1 -15325.194,E2 -15325.194} C_VEL
LIN {X 0,Y 318.449,Z 781.82,A -85,B 0,C 180,E1 -15326.191,E2 -15326.191} C_VEL
LIN {X 0,Y 318.759,Z 781.776,A -85,B 0,C 180,E1 -15329.014,E2 -15329.014} C_VEL
LIN {X 0,Y 319.11,Z 781.733,A -85,B 0,C 180,E1 -15331.907,E2 -15331.907} C_VEL
LIN {X 0,Y 319.468,Z 781.687,A -85,B 0,C 180,E1 -15335.515,E2 -15335.515} C_VEL
LIN {X 0,Y 319.527,Z 781.681,A -85,B 0,C 180,E1 -15338.013,E2 -15338.013} C_VEL
LIN {X 0,Y 319.521,Z 781.68,A -85,B 0,C 180,E1 -15341.596,E2 -15341.596} C_VEL
LIN {X 0,Y 319.483,Z 781.687,A -85,B 0,C 180,E1 -15345.256,E2 -15345.256} C_VEL
LIN {X 0,Y 319.523,Z 781.685,A -85,B 0,C 180,E1 -15348.711,E2 -15348.711} C_VEL
LIN {X 0,Y 319.547,Z 781.678,A -85,B 0,C 180,E1 -15352.349,E2 -15352.349} C_VEL
LIN {X 0,Y 319.553,Z 781.682,A -85,B 0,C 180,E1 -15355.122,E2 -15355.122} C_VEL
LIN {X 0,Y 319.517,Z 781.681,A -85,B 0,C 180,E1 -15358.136,E2 -15358.136} C_VEL
LIN {X 0,Y 319.564,Z 781.677,A -85,B 0,C 180,E1 -15361.602,E2 -15361.602} C_VEL
LIN {X 0,Y 319.567,Z 781.681,A -85,B 0,C 180,E1 -15365.301,E2 -15365.301} C_VEL
LIN {X 0,Y 319.559,Z 781.676,A -85,B 0,C 180,E1 -15368.045,E2 -15368.045} C_VEL
LIN {X 0,Y 319.605,Z 781.671,A -85,B 0,C 180,E1 -15372.07,E2 -15372.07} C_VEL
LIN {X 0,Y 319.723,Z 781.657,A -85,B 0,C 180,E1 -15376.007,E2 -15376.007} C_VEL
LIN {X 0,Y 319.726,Z 781.659,A -85,B 0,C 180,E1 -15379.872,E2 -15379.872} C_VEL
LIN {X 0,Y 319.887,Z 781.64,A -85,B 0,C 180,E1 -15383.693,E2 -15383.693} C_VEL
LIN {X 0,Y 319.944,Z 781.63,A -85,B 0,C 180,E1 -15387.482,E2 -15387.482} C_VEL
LIN {X 0,Y 319.986,Z 781.623,A -85,B 0,C 180,E1 -15391.259,E2 -15391.259} C_VEL
LIN {X 0,Y 319.702,Z 781.658,A -85,B 0,C 180,E1 -15395.045,E2 -15395.045} C_VEL
LIN {X 0,Y 319.842,Z 781.641,A -85,B 0,C 180,E1 -15397.576,E2 -15397.576} C_VEL
LIN {X 0,Y 319.702,Z 781.658,A -85,B 0,C 180,E1 -15401.411,E2 -15401.411} C_VEL
LIN {X 0,Y 319.703,Z 781.661,A -85,B 0,C 180,E1 -15404.711,E2 -15404.711} C_VEL
LIN {X 0,Y 319.605,Z 781.671,A -85,B 0,C 180,E1 -15407.93,E2 -15407.93} C_VEL
LIN {X 0,Y 319.559,Z 781.676,A -85,B 0,C 180,E1 -15411.955,E2 -15411.955} C_VEL
LIN {X 0,Y 319.562,Z 781.676,A -85,B 0,C 180,E1 -15416.095,E2 -15416.095} C_VEL
LIN {X 0,Y 319.535,Z 781.683,A -85,B 0,C 180,E1 -15418.939,E2 -15418.939} C_VEL
LIN {X 0,Y 319.517,Z 781.681,A -85,B 0,C 180,E1 -15421.864,E2 -15421.864} C_VEL
LIN {X 0,Y 319.573,Z 781.675,A -85,B 0,C 180,E1 -15425.544,E2 -15425.544} C_VEL
LIN {X 0,Y 319.552,Z 781.678,A -85,B 0,C 180,E1 -15429.67,E2 -15429.67} C_VEL
LIN {X 0,Y 319.516,Z 781.685,A -85,B 0,C 180,E1 -15433.462,E2 -15433.462} C_VEL
LIN {X 0,Y 319.549,Z 781.68,A -85,B 0,C 180,E1 -15437.018,E2 -15437.018} C_VEL
LIN {X 0,Y 319.541,Z 781.678,A -85,B 0,C 180,E1 -15440.372,E2 -15440.372} C_VEL
LIN {X 0,Y 319.513,Z 781.687,A -85,B 0,C 180,E1 -15443.568,E2 -15443.568} C_VEL
LIN {X 0,Y 319.307,Z 781.707,A -85,B 0,C 180,E1 -15446.761,E2 -15446.761} C_VEL
LIN {X 0,Y 319.029,Z 781.747,A -85,B 0,C 180,E1 -15449.559,E2 -15449.559} C_VEL
LIN {X 0,Y 318.672,Z 781.787,A -85,B 0,C 180,E1 -15452.412,E2 -15452.412} C_VEL
LIN {X 0,Y 318.28,Z 781.992,A -85,B 0,C 180,E1 -15455.37,E2 -15455.37} C_VEL
LIN {X 0,Y 318.282,Z 785.866,A -85,B 0,C 180,E1 -15459.186,E2 -15459.186} C_VEL
LIN {X 0,Y 321.008,Z 798.921,A -85,B 0,C 180,E1 -15459.981,E2 -15459.981} C_VEL
LIN {X 0,Y 323.593,Z 811.702,A -85,B 0,C 180,E1 -15460.989,E2 -15460.989} C_VEL
LIN {X 0,Y 324.211,Z 814.859,A -85,B 0,C 180,E1 -15461.274,E2 -15461.274} C_VEL
LIN {X 0,Y 324.233,Z 818.338,A -85,B 0,C 180,E1 -15461.584,E2 -15461.584} C_VEL
LIN {X 0,Y 322.87,Z 823.488,A -85,B 0,C 180,E1 -15462.033,E2 -15462.033} C_VEL
LIN {X 0,Y 317.266,Z 834.839,A -85,B 0,C 180,E1 -15463.14,E2 -15463.14} C_VEL
LIN {X 0,Y 315.607,Z 839.628,A -85,B 0,C 180,E1 -15463.73,E2 -15463.73} C_VEL
LIN {X 0,Y 315.373,Z 841.192,A -85,B 0,C 180,E1 -15463.95,E2 -15463.95} C_VEL
LIN {X 0,Y 314.354,Z 850.759,A -85,B 0,C 180,E1 -15465.434,E2 -15465.434} C_VEL
LIN {X 0,Y 313.393,Z 859.377,A -85,B 0,C 180,E1 -15467.042,E2 -15467.042} C_VEL
LIN {X 0,Y 312.538,Z 867.849,A -85,B 0,C 180,E1 -15468.982,E2 -15468.982} C_VEL
LIN {X 0,Y 311.828,Z 874.711,A -85,B 0,C 180,E1 -15470.924,E2 -15470.924} C_VEL
LIN {X 0,Y 311.458,Z 880.216,A -85,B 0,C 180,E1 -15472.873,E2 -15472.873} C_VEL
LIN {X 0,Y 311.173,Z 884.521,A -85,B 0,C 180,E1 -15474.818,E2 -15474.818} C_VEL
LIN {X 0,Y 311.033,Z 886.782,A -85,B 0,C 180,E1 -15476.114,E2 -15476.114} C_VEL
LIN {X 0,Y 310.972,Z 888.584,A -85,B 0,C 180,E1 -15477.411,E2 -15477.411} C_VEL
LIN {X 0,Y 310.965,Z 889.983,A -85,B 0,C 180,E1 -15478.706,E2 -15478.706} C_VEL
LIN {X 0,Y 310.999,Z 890.949,A -85,B 0,C 180,E1 -15480.001,E2 -15480.001} C_VEL
LIN {X 0,Y 311.099,Z 891.479,A -85,B 0,C 180,E1 -15481.296,E2 -15481.296} C_VEL
LIN {X 0,Y 311.273,Z 891.617,A -85,B 0,C 180,E1 -15482.589,E2 -15482.589} C_VEL
LIN {X 0,Y 311.453,Z 891.36,A -85,B 0,C 180,E1 -15483.883,E2 -15483.883} C_VEL
LIN {X 0,Y 311.742,Z 889.608,A -85,B 0,C 180,E1 -15486.474,E2 -15486.474} C_VEL
LIN {X 0,Y 312.642,Z 887.087,A -85,B 0,C 180,E1 -15488.468,E2 -15488.468} C_VEL
LIN {X 0,Y 313.46,Z 883.799,A -85,B 0,C 180,E1 -15490.334,E2 -15490.334} C_VEL
LIN {X 0,Y 314.541,Z 879.377,A -85,B 0,C 180,E1 -15492.256,E2 -15492.256} C_VEL
LIN {X 0,Y 316.284,Z 872.766,A -85,B 0,C 180,E1 -15494.478,E2 -15494.478} C_VEL
LIN {X 0,Y 318.295,Z 864.288,A -85,B 0,C 180,E1 -15496.682,E2 -15496.682} C_VEL
LIN {X 0,Y 320.574,Z 855.247,A -85,B 0,C 180,E1 -15498.536,E2 -15498.536} C_VEL
LIN {X 0,Y 322.726,Z 845.33,A -85,B 0,C 180,E1 -15500.199,E2 -15500.199} C_VEL
LIN {X 0,Y 325.1,Z 833.848,A -85,B 0,C 180,E1 -15501.73,E2 -15501.73} C_VEL
LIN {X 0,Y 326.104,Z 828.641,A -85,B 0,C 180,E1 -15502.325,E2 -15502.325} C_VEL
LIN {X 0,Y 325.24,Z 822.477,A -85,B 0,C 180,E1 -15503.255,E2 -15503.255} C_VEL
LIN {X 0,Y 322.058,Z 812.019,A -85,B 0,C 180,E1 -15504.965,E2 -15504.965} C_VEL
LIN {X 0,Y 317.925,Z 802.512,A -85,B 0,C 180,E1 -15506.676,E2 -15506.676} C_VEL
LIN {X 0,Y 313.609,Z 794.501,A -85,B 0,C 180,E1 -15508.306,E2 -15508.306} C_VEL
LIN {X 0,Y 313.42,Z 793.711,A -85,B 0,C 180,E1 -15508.441,E2 -15508.441} C_VEL
LIN {X 0,Y 313.69,Z 791.617,A -85,B 0,C 180,E1 -15511.639,E2 -15511.639} C_VEL
LIN {X 0,Y 313.834,Z 790.26,A -85,B 0,C 180,E1 -15514.047,E2 -15514.047} C_VEL
LIN {X 0,Y 313.825,Z 788.793,A -85,B 0,C 180,E1 -15517.205,E2 -15517.205} C_VEL
LIN {X 0,Y 313.732,Z 787.816,A -85,B 0,C 180,E1 -15520.516,E2 -15520.516} C_VEL
LIN {X 0,Y 313.679,Z 787.455,A -85,B 0,C 180,E1 -15524.195,E2 -15524.195} C_VEL
LIN {X 0,Y 313.554,Z 788.147,A -85,B 0,C 180,E1 -15527.196,E2 -15527.196} C_VEL
LIN {X 0,Y 314.683,Z 794.446,A -85,B 0,C 180,E1 -15531.416,E2 -15531.416} C_VEL
LIN {X 0,Y 314.989,Z 797.616,A -85,B 0,C 180,E1 -15533.441,E2 -15533.441} C_VEL
LIN {X 0,Y 314.502,Z 801.873,A -85,B 0,C 180,E1 -15536.037,E2 -15536.037} C_VEL
LIN {X 0,Y 313.532,Z 808.061,A -85,B 0,C 180,E1 -15539.712,E2 -15539.712} C_VEL
LIN {X 0,Y 313.131,Z 811.359,A -85,B 0,C 180,E1 -15541.618,E2 -15541.618} C_VEL
LIN {X 0,Y 313.798,Z 814.989,A -85,B 0,C 180,E1 -15542.029,E2 -15542.029} C_VEL
LIN {X 0,Y 314.942,Z 817.84,A -85,B 0,C 180,E1 -15542.479,E2 -15542.479} C_VEL
LIN {X 0,Y 315.783,Z 821.353,A -85,B 0,C 180,E1 -15542.904,E2 -15542.904} C_VEL
LIN {X 0,Y 317.487,Z 827.516,A -85,B 0,C 180,E1 -15543.722,E2 -15543.722} C_VEL
LIN {X 0,Y 319.936,Z 840.434,A -85,B 0,C 180,E1 -15545.331,E2 -15545.331} C_VEL
LIN {X 0,Y 321.164,Z 852.284,A -85,B 0,C 180,E1 -15546.803,E2 -15546.803} C_VEL
LIN {X 0,Y 320.949,Z 864.187,A -85,B 0,C 180,E1 -15548.314,E2 -15548.314} C_VEL
LIN {X 0,Y 320.208,Z 873.454,A -85,B 0,C 180,E1 -15549.609,E2 -15549.609} C_VEL
LIN {X 0,Y 318.256,Z 882.62,A -85,B 0,C 180,E1 -15550.991,E2 -15550.991} C_VEL
LIN {X 0,Y 316.103,Z 893.08,A -85,B 0,C 180,E1 -15552.901,E2 -15552.901} C_VEL
LIN {X 0,Y 314.44,Z 901.349,A -85,B 0,C 180,E1 -15554.774,E2 -15554.774} C_VEL
LIN {X 0,Y 312.859,Z 909.378,A -85,B 0,C 180,E1 -15557.018,E2 -15557.018} C_VEL
LIN {X 0,Y 311.926,Z 914.897,A -85,B 0,C 180,E1 -15558.959,E2 -15558.959} C_VEL
LIN {X 0,Y 311.338,Z 919.277,A -85,B 0,C 180,E1 -15560.908,E2 -15560.908} C_VEL
LIN {X 0,Y 311.051,Z 921.626,A -85,B 0,C 180,E1 -15562.209,E2 -15562.209} C_VEL
LIN {X 0,Y 310.893,Z 924.242,A -85,B 0,C 180,E1 -15564.083,E2 -15564.083} C_VEL
LIN {X 0,Y 310.879,Z 926.059,A -85,B 0,C 180,E1 -15566.111,E2 -15566.111} C_VEL
LIN {X 0,Y 311.085,Z 927.599,A -85,B 0,C 180,E1 -15568.705,E2 -15568.705} C_VEL
LIN {X 0,Y 311.112,Z 928.254,A -85,B 0,C 180,E1 -15570,E2 -15570} C_VEL
LIN {X 0,Y 310.988,Z 928.47,A -85,B 0,C 180,E1 -15571.295,E2 -15571.295} C_VEL
LIN {X 0,Y 310.821,Z 928.274,A -85,B 0,C 180,E1 -15572.592,E2 -15572.592} C_VEL
LIN {X 0,Y 310.848,Z 927.678,A -85,B 0,C 180,E1 -15573.889,E2 -15573.889} C_VEL
LIN {X 0,Y 310.844,Z 925.963,A -85,B 0,C 180,E1 -15575.83,E2 -15575.83} C_VEL
LIN {X 0,Y 311.156,Z 922.174,A -85,B 0,C 180,E1 -15578.442,E2 -15578.442} C_VEL
LIN {X 0,Y 311.688,Z 918.201,A -85,B 0,C 180,E1 -15580.392,E2 -15580.392} C_VEL
LIN {X 0,Y 312.493,Z 913.148,A -85,B 0,C 180,E1 -15582.337,E2 -15582.337} C_VEL
LIN {X 0,Y 314.004,Z 905.764,A -85,B 0,C 180,E1 -15584.584,E2 -15584.584} C_VEL
LIN {X 0,Y 315.509,Z 898.045,A -85,B 0,C 180,E1 -15586.494,E2 -15586.494} C_VEL
LIN {X 0,Y 317.518,Z 888.572,A -85,B 0,C 180,E1 -15588.386,E2 -15588.386} C_VEL
LIN {X 0,Y 320.061,Z 877.198,A -85,B 0,C 180,E1 -15590.233,E2 -15590.233} C_VEL
LIN {X 0,Y 321.134,Z 871.694,A -85,B 0,C 180,E1 -15591,E2 -15591} C_VEL
LIN {X 0,Y 322.018,Z 858.655,A -85,B 0,C 180,E1 -15592.729,E2 -15592.729} C_VEL
LIN {X 0,Y 321.529,Z 848.183,A -85,B 0,C 180,E1 -15594.059,E2 -15594.059} C_VEL
LIN {X 0,Y 319.555,Z 836.121,A -85,B 0,C 180,E1 -15595.613,E2 -15595.613} C_VEL
LIN {X 0,Y 316.282,Z 824.021,A -85,B 0,C 180,E1 -15597.272,E2 -15597.272} C_VEL
LIN {X 0,Y 313.659,Z 816.158,A -85,B 0,C 180,E1 -15598.413,E2 -15598.413} C_VEL
LIN {X 0,Y 313.544,Z 815.287,A -85,B 0,C 180,E1 -15598.529,E2 -15598.529} C_VEL
LIN {X 0,Y 314.637,Z 809.797,A -85,B 0,C 180,E1 -15602.418,E2 -15602.418} C_VEL
LIN {X 0,Y 315.474,Z 806.068,A -85,B 0,C 180,E1 -15605.396,E2 -15605.396} C_VEL
LIN {X 0,Y 315.744,Z 804.347,A -85,B 0,C 180,E1 -15606.94,E2 -15606.94} C_VEL
LIN {X 0,Y 315.824,Z 802.458,A -85,B 0,C 180,E1 -15608.843,E2 -15608.843} C_VEL
LIN {X 0,Y 315.581,Z 799.935,A -85,B 0,C 180,E1 -15611.921,E2 -15611.921} C_VEL
LIN {X 0,Y 315.222,Z 797.712,A -85,B 0,C 180,E1 -15615.517,E2 -15615.517} C_VEL
LIN {X 0,Y 314.88,Z 796.155,A -85,B 0,C 180,E1 -15619.365,E2 -15619.365} C_VEL
LIN {X 0,Y 314.581,Z 795.421,A -85,B 0,C 180,E1 -15622.899,E2 -15622.899} C_VEL
LIN {X 0,Y 314.24,Z 795.293,A -85,B 0,C 180,E1 -15626.003,E2 -15626.003} C_VEL
LIN {X 0,Y 313.805,Z 795.593,A -85,B 0,C 180,E1 -15628.994,E2 -15628.994} C_VEL
LIN {X 0,Y 313.404,Z 796.149,A -85,B 0,C 180,E1 -15631.638,E2 -15631.638} C_VEL
LIN {X 0,Y 314.06,Z 798.181,A -85,B 0,C 180,E1 -15631.969,E2 -15631.969} C_VEL
LIN {X 0,Y 316.193,Z 801.554,A -85,B 0,C 180,E1 -15632.758,E2 -15632.758} C_VEL
LIN {X 0,Y 320.879,Z 810.895,A -85,B 0,C 180,E1 -15634.607,E2 -15634.607} C_VEL
LIN {X 0,Y 324.496,Z 820.686,A -85,B 0,C 180,E1 -15636.33,E2 -15636.33} C_VEL
LIN {X 0,Y 326.154,Z 827.996,A -85,B 0,C 180,E1 -15637.512,E2 -15637.512} C_VEL
LIN {X 0,Y 326.291,Z 829.162,A -85,B 0,C 180,E1 -15637.689,E2 -15637.689} C_VEL
LIN {X 0,Y 323.971,Z 841.265,A -85,B 0,C 180,E1 -15639.192,E2 -15639.192} C_VEL
LIN {X 0,Y 321.578,Z 852.179,A -85,B 0,C 180,E1 -15640.862,E2 -15640.862} C_VEL
LIN {X 0,Y 319.159,Z 861.796,A -85,B 0,C 180,E1 -15642.705,E2 -15642.705} C_VEL
LIN {X 0,Y 317.291,Z 869.694,A -85,B 0,C 180,E1 -15644.584,E2 -15644.584} C_VEL
LIN {X 0,Y 315.647,Z 876.12,A -85,B 0,C 180,E1 -15646.479,E2 -15646.479} C_VEL
LIN {X 0,Y 314.221,Z 881.289,A -85,B 0,C 180,E1 -15648.386,E2 -15648.386} C_VEL
LIN {X 0,Y 313.272,Z 885.362,A -85,B 0,C 180,E1 -15650.312,E2 -15650.312} C_VEL
LIN {X 0,Y 312.35,Z 888.45,A -85,B 0,C 180,E1 -15652.24,E2 -15652.24} C_VEL
LIN {X 0,Y 311.765,Z 889.96,A -85,B 0,C 180,E1 -15653.527,E2 -15653.527} C_VEL
LIN {X 0,Y 311.665,Z 891.032,A -85,B 0,C 180,E1 -15654.824,E2 -15654.824} C_VEL
LIN {X 0,Y 311.541,Z 891.731,A -85,B 0,C 180,E1 -15656.118,E2 -15656.118} C_VEL
LIN {X 0,Y 311.305,Z 892.02,A -85,B 0,C 180,E1 -15657.411,E2 -15657.411} C_VEL
LIN {X 0,Y 311.139,Z 891.901,A -85,B 0,C 180,E1 -15658.704,E2 -15658.704} C_VEL
LIN {X 0,Y 311.046,Z 891.386,A -85,B 0,C 180,E1 -15659.999,E2 -15659.999} C_VEL
LIN {X 0,Y 311.005,Z 890.47,A -85,B 0,C 180,E1 -15661.294,E2 -15661.294} C_VEL
LIN {X 0,Y 310.988,Z 889.102,A -85,B 0,C 180,E1 -15662.589,E2 -15662.589} C_VEL
LIN {X 0,Y 311.136,Z 886.269,A -85,B 0,C 180,E1 -15664.533,E2 -15664.533} C_VEL
LIN {X 0,Y 311.363,Z 881.877,A -85,B 0,C 180,E1 -15666.706,E2 -15666.706} C_VEL
LIN {X 0,Y 311.678,Z 877.402,A -85,B 0,C 180,E1 -15668.427,E2 -15668.427} C_VEL
LIN {X 0,Y 312.409,Z 869.95,A -85,B 0,C 180,E1 -15670.694,E2 -15670.694} C_VEL
LIN {X 0,Y 313.223,Z 861.868,A -85,B 0,C 180,E1 -15672.635,E2 -15672.635} C_VEL
LIN {X 0,Y 314.353,Z 851.923,A -85,B 0,C 180,E1 -15674.566,E2 -15674.566} C_VEL
LIN {X 0,Y 315.487,Z 841.695,A -85,B 0,C 180,E1 -15676.167,E2 -15676.167} C_VEL
LIN {X 0,Y 316.469,Z 830.401,A -85,B 0,C 180,E1 -15677.611,E2 -15677.611} C_VEL
LIN {X 0,Y 317.415,Z 819.641,A -85,B 0,C 180,E1 -15678.725,E2 -15678.725} C_VEL
LIN {X 0,Y 317.559,Z 817.864,A -85,B 0,C 180,E1 -15678.884,E2 -15678.884} C_VEL
LIN {X 0,Y 315.074,Z 805.345,A -85,B 0,C 180,E1 -15680.01,E2 -15680.01} C_VEL
LIN {X 0,Y 312.363,Z 792.379,A -85,B 0,C 180,E1 -15680.934,E2 -15680.934} C_VEL
LIN {X 0,Y 311.261,Z 786.892,A -85,B 0,C 180,E1 -15681.25,E2 -15681.25} C_VEL
LIN {X 0,Y 311.372,Z 783.138,A -85,B 0,C 180,E1 -15685.465,E2 -15685.465} C_VEL
LIN {X 0,Y 311.493,Z 782.686,A -85,B 0,C 180,E1 -15686.822,E2 -15686.822} C_VEL
LIN {X 0,Y 311.786,Z 782.645,A -85,B 0,C 180,E1 -15689.728,E2 -15689.728} C_VEL
LIN {X 0,Y 312.267,Z 782.584,A -85,B 0,C 180,E1 -15693.619,E2 -15693.619} C_VEL
LIN {X 0,Y 312.45,Z 782.562,A -85,B 0,C 180,E1 -15695.928,E2 -15695.928} C_VEL
LIN {X 0,Y 312.489,Z 782.558,A -85,B 0,C 180,E1 -15699.028,E2 -15699.028} C_VEL
LIN {X 0,Y 312.485,Z 782.56,A -85,B 0,C 180,E1 -15702.43,E2 -15702.43} C_VEL
LIN {X 0,Y 312.452,Z 782.561,A -85,B 0,C 180,E1 -15706.034,E2 -15706.034} C_VEL
LIN {X 0,Y 312.498,Z 782.555,A -85,B 0,C 180,E1 -15709.873,E2 -15709.873} C_VEL
LIN {X 0,Y 312.529,Z 782.552,A -85,B 0,C 180,E1 -15714.049,E2 -15714.049} C_VEL
LIN {X 0,Y 312.494,Z 782.559,A -85,B 0,C 180,E1 -15717.332,E2 -15717.332} C_VEL
LIN {X 0,Y 312.5,Z 782.56,A -85,B 0,C 180,E1 -15721.29,E2 -15721.29} C_VEL
LIN {X 0,Y 312.54,Z 782.551,A -85,B 0,C 180,E1 -15724.707,E2 -15724.707} C_VEL
LIN {X 0,Y 312.555,Z 782.552,A -85,B 0,C 180,E1 -15727.526,E2 -15727.526} C_VEL
LIN {X 0,Y 312.558,Z 782.552,A -85,B 0,C 180,E1 -15731.651,E2 -15731.651} C_VEL
LIN {X 0,Y 312.677,Z 782.538,A -85,B 0,C 180,E1 -15735.685,E2 -15735.685} C_VEL
LIN {X 0,Y 312.676,Z 782.538,A -85,B 0,C 180,E1 -15739.641,E2 -15739.641} C_VEL
LIN {X 0,Y 312.786,Z 782.521,A -85,B 0,C 180,E1 -15742.252,E2 -15742.252} C_VEL
LIN {X 0,Y 312.675,Z 782.533,A -85,B 0,C 180,E1 -15744.842,E2 -15744.842} C_VEL
LIN {X 0,Y 312.956,Z 782.499,A -85,B 0,C 180,E1 -15748.713,E2 -15748.713} C_VEL
LIN {X 0,Y 312.955,Z 782.499,A -85,B 0,C 180,E1 -15751.287,E2 -15751.287} C_VEL
LIN {X 0,Y 312.829,Z 782.517,A -85,B 0,C 180,E1 -15756.45,E2 -15756.45} C_VEL
LIN {X 0,Y 312.741,Z 782.525,A -85,B 0,C 180,E1 -15759.051,E2 -15759.051} C_VEL
LIN {X 0,Y 312.623,Z 782.54,A -85,B 0,C 180,E1 -15762.992,E2 -15762.992} C_VEL
LIN {X 0,Y 312.613,Z 782.541,A -85,B 0,C 180,E1 -15765.651,E2 -15765.651} C_VEL
LIN {X 0,Y 312.53,Z 782.551,A -85,B 0,C 180,E1 -15769.713,E2 -15769.713} C_VEL
LIN {X 0,Y 312.514,Z 782.558,A -85,B 0,C 180,E1 -15772.78,E2 -15772.78} C_VEL
LIN {X 0,Y 312.522,Z 782.553,A -85,B 0,C 180,E1 -15775.909,E2 -15775.909} C_VEL
LIN {X 0,Y 312.488,Z 782.557,A -85,B 0,C 180,E1 -15779.656,E2 -15779.656} C_VEL
LIN {X 0,Y 312.512,Z 782.554,A -85,B 0,C 180,E1 -15783.69,E2 -15783.69} C_VEL
LIN {X 0,Y 312.513,Z 782.556,A -85,B 0,C 180,E1 -15787.387,E2 -15787.387} C_VEL
LIN {X 0,Y 312.484,Z 782.559,A -85,B 0,C 180,E1 -15790.71,E2 -15790.71} C_VEL
LIN {X 0,Y 312.446,Z 782.562,A -85,B 0,C 180,E1 -15794.211,E2 -15794.211} C_VEL
LIN {X 0,Y 312.479,Z 782.558,A -85,B 0,C 180,E1 -15797.92,E2 -15797.92} C_VEL
LIN {X 0,Y 312.49,Z 782.558,A -85,B 0,C 180,E1 -15800.972,E2 -15800.972} C_VEL
LIN {X 0,Y 312.448,Z 782.562,A -85,B 0,C 180,E1 -15804.211,E2 -15804.211} C_VEL
LIN {X 0,Y 312.202,Z 782.595,A -85,B 0,C 180,E1 -15807.3,E2 -15807.3} C_VEL
LIN {X 0,Y 311.865,Z 782.635,A -85,B 0,C 180,E1 -15810.281,E2 -15810.281} C_VEL
LIN {X 0,Y 311.507,Z 782.68,A -85,B 0,C 180,E1 -15813.179,E2 -15813.179} C_VEL
LIN {X 0,Y 311.211,Z 782.791,A -85,B 0,C 180,E1 -15815.485,E2 -15815.485} C_VEL
LIN {X 0,Y 311.235,Z 786.248,A -85,B 0,C 180,E1 -15818.899,E2 -15818.899} C_VEL
LIN {X 0,Y 313.96,Z 799.553,A -85,B 0,C 180,E1 -15819.732,E2 -15819.732} C_VEL
LIN {X 0,Y 316.613,Z 812.693,A -85,B 0,C 180,E1 -15820.806,E2 -15820.806} C_VEL
LIN {X 0,Y 317.419,Z 817.668,A -85,B 0,C 180,E1 -15821.275,E2 -15821.275} C_VEL
LIN {X 0,Y 316.424,Z 829.226,A -85,B 0,C 180,E1 -15822.437,E2 -15822.437} C_VEL
LIN {X 0,Y 315.442,Z 840.362,A -85,B 0,C 180,E1 -15823.831,E2 -15823.831} C_VEL
LIN {X 0,Y 315.373,Z 841.192,A -85,B 0,C 180,E1 -15823.95,E2 -15823.95} C_VEL
LIN {X 0,Y 314.301,Z 845.793,A -85,B 0,C 180,E1 -15824.608,E2 -15824.608} C_VEL
LIN {X 0,Y 310.684,Z 852.88,A -85,B 0,C 180,E1 -15825.703,E2 -15825.703} C_VEL
LIN {X 0,Y 307.057,Z 859.464,A -85,B 0,C 180,E1 -15826.904,E2 -15826.904} C_VEL
LIN {X 0,Y 305.98,Z 863.252,A -85,B 0,C 180,E1 -15827.718,E2 -15827.718} C_VEL
LIN {X 0,Y 305.146,Z 871.115,A -85,B 0,C 180,E1 -15829.719,E2 -15829.719} C_VEL
LIN {X 0,Y 304.505,Z 878.346,A -85,B 0,C 180,E1 -15832.042,E2 -15832.042} C_VEL
LIN {X 0,Y 304.168,Z 882.842,A -85,B 0,C 180,E1 -15833.88,E2 -15833.88} C_VEL
LIN {X 0,Y 303.967,Z 886.9,A -85,B 0,C 180,E1 -15836.024,E2 -15836.024} C_VEL
LIN {X 0,Y 303.886,Z 888.776,A -85,B 0,C 180,E1 -15837.35,E2 -15837.35} C_VEL
LIN {X 0,Y 303.87,Z 890.238,A -85,B 0,C 180,E1 -15838.676,E2 -15838.676} C_VEL
LIN {X 0,Y 303.908,Z 891.299,A -85,B 0,C 180,E1 -15840.001,E2 -15840.001} C_VEL
LIN {X 0,Y 304.014,Z 891.911,A -85,B 0,C 180,E1 -15841.326,E2 -15841.326} C_VEL
LIN {X 0,Y 304.195,Z 892.112,A -85,B 0,C 180,E1 -15842.65,E2 -15842.65} C_VEL
LIN {X 0,Y 304.38,Z 891.93,A -85,B 0,C 180,E1 -15843.973,E2 -15843.973} C_VEL
LIN {X 0,Y 304.482,Z 891.366,A -85,B 0,C 180,E1 -15845.299,E2 -15845.299} C_VEL
LIN {X 0,Y 304.734,Z 890.355,A -85,B 0,C 180,E1 -15846.623,E2 -15846.623} C_VEL
LIN {X 0,Y 305.692,Z 887.957,A -85,B 0,C 180,E1 -15848.662,E2 -15848.662} C_VEL
LIN {X 0,Y 306.916,Z 883.564,A -85,B 0,C 180,E1 -15851.225,E2 -15851.225} C_VEL
LIN {X 0,Y 308.187,Z 878.945,A -85,B 0,C 180,E1 -15853.183,E2 -15853.183} C_VEL
LIN {X 0,Y 310.135,Z 872.022,A -85,B 0,C 180,E1 -15855.444,E2 -15855.444} C_VEL
LIN {X 0,Y 312.071,Z 864.722,A -85,B 0,C 180,E1 -15857.363,E2 -15857.363} C_VEL
LIN {X 0,Y 314.495,Z 855.658,A -85,B 0,C 180,E1 -15859.247,E2 -15859.247} C_VEL
LIN {X 0,Y 317.061,Z 844.911,A -85,B 0,C 180,E1 -15861.071,E2 -15861.071} C_VEL
LIN {X 0,Y 319.624,Z 833.259,A -85,B 0,C 180,E1 -15862.632,E2 -15862.632} C_VEL
LIN {X 0,Y 320.168,Z 830.65,A -85,B 0,C 180,E1 -15862.932,E2 -15862.932} C_VEL
LIN {X 0,Y 319.265,Z 824.661,A -85,B 0,C 180,E1 -15863.911,E2 -15863.911} C_VEL
LIN {X 0,Y 316.64,Z 815.591,A -85,B 0,C 180,E1 -15865.51,E2 -15865.51} C_VEL
LIN {X 0,Y 313.179,Z 807.127,A -85,B 0,C 180,E1 -15867.157,E2 -15867.157} C_VEL
LIN {X 0,Y 309.405,Z 799.567,A -85,B 0,C 180,E1 -15868.799,E2 -15868.799} C_VEL
LIN {X 0,Y 307.305,Z 796.405,A -85,B 0,C 180,E1 -15869.651,E2 -15869.651} C_VEL
LIN {X 0,Y 306.695,Z 794.668,A -85,B 0,C 180,E1 -15870.007,E2 -15870.007} C_VEL
LIN {X 0,Y 306.91,Z 793.434,A -85,B 0,C 180,E1 -15872.083,E2 -15872.083} C_VEL
LIN {X 0,Y 307.075,Z 792.02,A -85,B 0,C 180,E1 -15874.903,E2 -15874.903} C_VEL
LIN {X 0,Y 307.108,Z 790.829,A -85,B 0,C 180,E1 -15878.163,E2 -15878.163} C_VEL
LIN {X 0,Y 307.05,Z 790.156,A -85,B 0,C 180,E1 -15881.59,E2 -15881.59} C_VEL
LIN {X 0,Y 307.052,Z 790.256,A -85,B 0,C 180,E1 -15884.802,E2 -15884.802} C_VEL
LIN {X 0,Y 307.014,Z 790.862,A -85,B 0,C 180,E1 -15887.1,E2 -15887.1} C_VEL
LIN {X 0,Y 307.017,Z 791.884,A -85,B 0,C 180,E1 -15889.063,E2 -15889.063} C_VEL
LIN {X 0,Y 307.765,Z 796.137,A -85,B 0,C 180,E1 -15891.934,E2 -15891.934} C_VEL
LIN {X 0,Y 307.894,Z 798.704,A -85,B 0,C 180,E1 -15893.596,E2 -15893.596} C_VEL
LIN {X 0,Y 307.224,Z 803.702,A -85,B 0,C 180,E1 -15896.7,E2 -15896.7} C_VEL
LIN {X 0,Y 306.406,Z 809.243,A -85,B 0,C 180,E1 -15899.947,E2 -15899.947} C_VEL
LIN {X 0,Y 307.202,Z 813.117,A -85,B 0,C 180,E1 -15900.465,E2 -15900.465} C_VEL
LIN {X 0,Y 308.461,Z 816.168,A -85,B 0,C 180,E1 -15901.016,E2 -15901.016} C_VEL
LIN {X 0,Y 309.658,Z 820.706,A -85,B 0,C 180,E1 -15901.664,E2 -15901.664} C_VEL
LIN {X 0,Y 312.018,Z 830.245,A -85,B 0,C 180,E1 -15903.026,E2 -15903.026} C_VEL
LIN {X 0,Y 314.068,Z 842.06,A -85,B 0,C 180,E1 -15904.621,E2 -15904.621} C_VEL
LIN {X 0,Y 315.018,Z 852.689,A -85,B 0,C 180,E1 -15906.032,E2 -15906.032} C_VEL
LIN {X 0,Y 314.863,Z 862.409,A -85,B 0,C 180,E1 -15907.327,E2 -15907.327} C_VEL
LIN {X 0,Y 313.909,Z 873.856,A -85,B 0,C 180,E1 -15909.009,E2 -15909.009} C_VEL
LIN {X 0,Y 311.654,Z 883.797,A -85,B 0,C 180,E1 -15910.572,E2 -15910.572} C_VEL
LIN {X 0,Y 309.736,Z 892.17,A -85,B 0,C 180,E1 -15912.163,E2 -15912.163} C_VEL
LIN {X 0,Y 307.875,Z 900.607,A -85,B 0,C 180,E1 -15914.102,E2 -15914.102} C_VEL
LIN {X 0,Y 306.164,Z 908.626,A -85,B 0,C 180,E1 -15916.391,E2 -15916.391} C_VEL
LIN {X 0,Y 304.941,Z 914.985,A -85,B 0,C 180,E1 -15918.703,E2 -15918.703} C_VEL
LIN {X 0,Y 304.289,Z 919.235,A -85,B 0,C 180,E1 -15920.696,E2 -15920.696} C_VEL
LIN {X 0,Y 303.848,Z 923.298,A -85,B 0,C 180,E1 -15923.359,E2 -15923.359} C_VEL
LIN {X 0,Y 303.801,Z 924.722,A -85,B 0,C 180,E1 -15924.691,E2 -15924.691} C_VEL
LIN {X 0,Y 303.787,Z 925.683,A -85,B 0,C 180,E1 -15926.02,E2 -15926.02} C_VEL
LIN {X 0,Y 304.026,Z 926.94,A -85,B 0,C 180,E1 -15928.675,E2 -15928.675} C_VEL
LIN {X 0,Y 304.055,Z 927.695,A -85,B 0,C 180,E1 -15930,E2 -15930} C_VEL
LIN {X 0,Y 303.896,Z 927.97,A -85,B 0,C 180,E1 -15931.325,E2 -15931.325} C_VEL
LIN {X 0,Y 303.754,Z 927.28,A -85,B 0,C 180,E1 -15933.98,E2 -15933.98} C_VEL
LIN {X 0,Y 303.741,Z 925.888,A -85,B 0,C 180,E1 -15935.757,E2 -15935.757} C_VEL
LIN {X 0,Y 303.995,Z 923.122,A -85,B 0,C 180,E1 -15937.973,E2 -15937.973} C_VEL
LIN {X 0,Y 304.449,Z 919.599,A -85,B 0,C 180,E1 -15939.97,E2 -15939.97} C_VEL
LIN {X 0,Y 305.556,Z 913.33,A -85,B 0,C 180,E1 -15942.621,E2 -15942.621} C_VEL
LIN {X 0,Y 307.143,Z 906.152,A -85,B 0,C 180,E1 -15944.917,E2 -15944.917} C_VEL
LIN {X 0,Y 309.082,Z 897.217,A -85,B 0,C 180,E1 -15947.193,E2 -15947.193} C_VEL
LIN {X 0,Y 311.235,Z 887.86,A -85,B 0,C 180,E1 -15949.113,E2 -15949.113} C_VEL
LIN {X 0,Y 314.002,Z 876.471,A -85,B 0,C 180,E1 -15950.984,E2 -15950.984} C_VEL
LIN {X 0,Y 315.048,Z 869.962,A -85,B 0,C 180,E1 -15951.941,E2 -15951.941} C_VEL
LIN {X 0,Y 315.899,Z 857.902,A -85,B 0,C 180,E1 -15953.607,E2 -15953.607} C_VEL
LIN {X 0,Y 315.252,Z 847.233,A -85,B 0,C 180,E1 -15955.06,E2 -15955.06} C_VEL
LIN {X 0,Y 313.31,Z 835.847,A -85,B 0,C 180,E1 -15956.656,E2 -15956.656} C_VEL
LIN {X 0,Y 310.189,Z 824.266,A -85,B 0,C 180,E1 -15958.412,E2 -15958.412} C_VEL
LIN {X 0,Y 308.836,Z 819.826,A -85,B 0,C 180,E1 -15959.12,E2 -15959.12} C_VEL
LIN {X 0,Y 307.246,Z 816.222,A -85,B 0,C 180,E1 -15959.789,E2 -15959.789} C_VEL
LIN {X 0,Y 306.919,Z 814.283,A -85,B 0,C 180,E1 -15960.071,E2 -15960.071} C_VEL
LIN {X 0,Y 307.879,Z 810.104,A -85,B 0,C 180,E1 -15963.22,E2 -15963.22} C_VEL
LIN {X 0,Y 308.365,Z 808.107,A -85,B 0,C 180,E1 -15964.865,E2 -15964.865} C_VEL
LIN {X 0,Y 308.794,Z 805.553,A -85,B 0,C 180,E1 -15967.193,E2 -15967.193} C_VEL
LIN {X 0,Y 308.843,Z 803.325,A -85,B 0,C 180,E1 -15969.581,E2 -15969.581} C_VEL
LIN {X 0,Y 308.732,Z 801.938,A -85,B 0,C 180,E1 -15971.312,E2 -15971.312} C_VEL
LIN {X 0,Y 308.361,Z 799.553,A -85,B 0,C 180,E1 -15975.045,E2 -15975.045} C_VEL
LIN {X 0,Y 307.994,Z 797.909,A -85,B 0,C 180,E1 -15978.852,E2 -15978.852} C_VEL
LIN {X 0,Y 307.738,Z 797.14,A -85,B 0,C 180,E1 -15981.929,E2 -15981.929} C_VEL
LIN {X 0,Y 307.385,Z 796.826,A -85,B 0,C 180,E1 -15985.396,E2 -15985.396} C_VEL
LIN {X 0,Y 307.004,Z 796.971,A -85,B 0,C 180,E1 -15988.228,E2 -15988.228} C_VEL
LIN {X 0,Y 306.693,Z 797.331,A -85,B 0,C 180,E1 -15990.084,E2 -15990.084} C_VEL
LIN {X 0,Y 307.745,Z 800.01,A -85,B 0,C 180,E1 -15990.64,E2 -15990.64} C_VEL
LIN {X 0,Y 309.296,Z 801.921,A -85,B 0,C 180,E1 -15991.246,E2 -15991.246} C_VEL
LIN {X 0,Y 310.743,Z 804.847,A -85,B 0,C 180,E1 -15991.892,E2 -15991.892} C_VEL
LIN {X 0,Y 313.632,Z 810.208,A -85,B 0,C 180,E1 -15993.135,E2 -15993.135} C_VEL
LIN {X 0,Y 317.707,Z 820.333,A -85,B 0,C 180,E1 -15995.145,E2 -15995.145} C_VEL
LIN {X 0,Y 319.767,Z 827.85,A -85,B 0,C 180,E1 -15996.51,E2 -15996.51} C_VEL
LIN {X 0,Y 320.221,Z 832.084,A -85,B 0,C 180,E1 -15997.189,E2 -15997.189} C_VEL
LIN {X 0,Y 317.643,Z 844.04,A -85,B 0,C 180,E1 -15998.757,E2 -15998.757} C_VEL
LIN {X 0,Y 315.124,Z 854.342,A -85,B 0,C 180,E1 -16000.455,E2 -16000.455} C_VEL
LIN {X 0,Y 312.61,Z 863.719,A -85,B 0,C 180,E1 -16002.331,E2 -16002.331} C_VEL
LIN {X 0,Y 310.64,Z 871.252,A -85,B 0,C 180,E1 -16004.246,E2 -16004.246} C_VEL
LIN {X 0,Y 308.883,Z 877.441,A -85,B 0,C 180,E1 -16006.177,E2 -16006.177} C_VEL
LIN {X 0,Y 307.384,Z 882.461,A -85,B 0,C 180,E1 -16008.124,E2 -16008.124} C_VEL
LIN {X 0,Y 306.347,Z 886.353,A -85,B 0,C 180,E1 -16010.091,E2 -16010.091} C_VEL
LIN {X 0,Y 305.388,Z 889.278,A -85,B 0,C 180,E1 -16012.062,E2 -16012.062} C_VEL
LIN {X 0,Y 304.756,Z 890.727,A -85,B 0,C 180,E1 -16013.377,E2 -16013.377} C_VEL
LIN {X 0,Y 304.628,Z 891.737,A -85,B 0,C 180,E1 -16014.704,E2 -16014.704} C_VEL
LIN {X 0,Y 304.484,Z 892.328,A -85,B 0,C 180,E1 -16016.028,E2 -16016.028} C_VEL
LIN {X 0,Y 304.244,Z 892.53,A -85,B 0,C 180,E1 -16017.351,E2 -16017.351} C_VEL
LIN {X 0,Y 303.956,Z 891.767,A -85,B 0,C 180,E1 -16019.999,E2 -16019.999} C_VEL
LIN {X 0,Y 303.91,Z 890.744,A -85,B 0,C 180,E1 -16021.324,E2 -16021.324} C_VEL
LIN {X 0,Y 303.902,Z 889.305,A -85,B 0,C 180,E1 -16022.65,E2 -16022.65} C_VEL
LIN {X 0,Y 304.055,Z 886.345,A -85,B 0,C 180,E1 -16024.639,E2 -16024.639} C_VEL
LIN {X 0,Y 304.282,Z 882.189,A -85,B 0,C 180,E1 -16026.698,E2 -16026.698} C_VEL
LIN {X 0,Y 304.625,Z 877.194,A -85,B 0,C 180,E1 -16028.623,E2 -16028.623} C_VEL
LIN {X 0,Y 305.29,Z 870.771,A -85,B 0,C 180,E1 -16030.611,E2 -16030.611} C_VEL
LIN {X 0,Y 306.115,Z 862.826,A -85,B 0,C 180,E1 -16032.596,E2 -16032.596} C_VEL
LIN {X 0,Y 307.225,Z 853.015,A -85,B 0,C 180,E1 -16034.573,E2 -16034.573} C_VEL
LIN {X 0,Y 308.357,Z 843.186,A -85,B 0,C 180,E1 -16036.184,E2 -16036.184} C_VEL
LIN {X 0,Y 309.379,Z 831.88,A -85,B 0,C 180,E1 -16037.686,E2 -16037.686} C_VEL
LIN {X 0,Y 310.479,Z 819.704,A -85,B 0,C 180,E1 -16038.988,E2 -16038.988} C_VEL
LIN {X 0,Y 310.108,Z 815.928,A -85,B 0,C 180,E1 -16039.355,E2 -16039.355} C_VEL
LIN {X 0,Y 307.571,Z 803.393,A -85,B 0,C 180,E1 -16040.47,E2 -16040.47} C_VEL
LIN {X 0,Y 304.681,Z 789.752,A -85,B 0,C 180,E1 -16041.412,E2 -16041.412} C_VEL
LIN {X 0,Y 304.197,Z 787.263,A -85,B 0,C 180,E1 -16041.565,E2 -16041.565} C_VEL
LIN {X 0,Y 304.323,Z 783.59,A -85,B 0,C 180,E1 -16045.754,E2 -16045.754} C_VEL
LIN {X 0,Y 304.651,Z 783.533,A -85,B 0,C 180,E1 -16048.975,E2 -16048.975} C_VEL
LIN {X 0,Y 305.01,Z 783.49,A -85,B 0,C 180,E1 -16052.001,E2 -16052.001} C_VEL
LIN {X 0,Y 305.305,Z 783.452,A -85,B 0,C 180,E1 -16055.132,E2 -16055.132} C_VEL
LIN {X 0,Y 305.429,Z 783.441,A -85,B 0,C 180,E1 -16058.524,E2 -16058.524} C_VEL
LIN {X 0,Y 305.436,Z 783.435,A -85,B 0,C 180,E1 -16061.855,E2 -16061.855} C_VEL
LIN {X 0,Y 305.394,Z 783.441,A -85,B 0,C 180,E1 -16065.51,E2 -16065.51} C_VEL
LIN {X 0,Y 305.435,Z 783.435,A -85,B 0,C 180,E1 -16068.142,E2 -16068.142} C_VEL
LIN {X 0,Y 305.461,Z 783.433,A -85,B 0,C 180,E1 -16071.595,E2 -16071.595} C_VEL
LIN {X 0,Y 305.455,Z 783.437,A -85,B 0,C 180,E1 -16074.886,E2 -16074.886} C_VEL
LIN {X 0,Y 305.434,Z 783.435,A -85,B 0,C 180,E1 -16078.357,E2 -16078.357} C_VEL
LIN {X 0,Y 305.469,Z 783.436,A -85,B 0,C 180,E1 -16081.108,E2 -16081.108} C_VEL
LIN {X 0,Y 305.493,Z 783.428,A -85,B 0,C 180,E1 -16084.081,E2 -16084.081} C_VEL
LIN {X 0,Y 305.484,Z 783.431,A -85,B 0,C 180,E1 -16086.977,E2 -16086.977} C_VEL
LIN {X 0,Y 305.509,Z 783.429,A -85,B 0,C 180,E1 -16091.212,E2 -16091.212} C_VEL
LIN {X 0,Y 305.617,Z 783.416,A -85,B 0,C 180,E1 -16095.347,E2 -16095.347} C_VEL
LIN {X 0,Y 305.615,Z 783.416,A -85,B 0,C 180,E1 -16099.399,E2 -16099.399} C_VEL
LIN {X 0,Y 305.736,Z 783.401,A -85,B 0,C 180,E1 -16102.072,E2 -16102.072} C_VEL
LIN {X 0,Y 305.646,Z 783.409,A -85,B 0,C 180,E1 -16104.723,E2 -16104.723} C_VEL
LIN {X 0,Y 305.925,Z 783.375,A -85,B 0,C 180,E1 -16108.684,E2 -16108.684} C_VEL
LIN {X 0,Y 305.923,Z 783.375,A -85,B 0,C 180,E1 -16111.316,E2 -16111.316} C_VEL
LIN {X 0,Y 305.774,Z 783.395,A -85,B 0,C 180,E1 -16116.599,E2 -16116.599} C_VEL
LIN {X 0,Y 305.684,Z 783.404,A -85,B 0,C 180,E1 -16119.261,E2 -16119.261} C_VEL
LIN {X 0,Y 305.576,Z 783.417,A -85,B 0,C 180,E1 -16123.297,E2 -16123.297} C_VEL
LIN {X 0,Y 305.542,Z 783.424,A -85,B 0,C 180,E1 -16126.023,E2 -16126.023} C_VEL
LIN {X 0,Y 305.476,Z 783.432,A -85,B 0,C 180,E1 -16130.188,E2 -16130.188} C_VEL
LIN {X 0,Y 305.478,Z 783.432,A -85,B 0,C 180,E1 -16133.04,E2 -16133.04} C_VEL
LIN {X 0,Y 305.461,Z 783.433,A -85,B 0,C 180,E1 -16136.198,E2 -16136.198} C_VEL
LIN {X 0,Y 305.441,Z 783.438,A -85,B 0,C 180,E1 -16139.035,E2 -16139.035} C_VEL
LIN {X 0,Y 305.429,Z 783.435,A -85,B 0,C 180,E1 -16141.954,E2 -16141.954} C_VEL
LIN {X 0,Y 305.455,Z 783.437,A -85,B 0,C 180,E1 -16145.114,E2 -16145.114} C_VEL
LIN {X 0,Y 305.434,Z 783.437,A -85,B 0,C 180,E1 -16148.528,E2 -16148.528} C_VEL
LIN {X 0,Y 305.449,Z 783.434,A -85,B 0,C 180,E1 -16152.587,E2 -16152.587} C_VEL
LIN {X 0,Y 305.42,Z 783.437,A -85,B 0,C 180,E1 -16156.346,E2 -16156.346} C_VEL
LIN {X 0,Y 305.453,Z 783.434,A -85,B 0,C 180,E1 -16159.894,E2 -16159.894} C_VEL
LIN {X 0,Y 305.414,Z 783.442,A -85,B 0,C 180,E1 -16163.649,E2 -16163.649} C_VEL
LIN {X 0,Y 305.234,Z 783.46,A -85,B 0,C 180,E1 -16166.456,E2 -16166.456} C_VEL
LIN {X 0,Y 304.907,Z 783.505,A -85,B 0,C 180,E1 -16169.531,E2 -16169.531} C_VEL
LIN {X 0,Y 304.527,Z 783.549,A -85,B 0,C 180,E1 -16172.513,E2 -16172.513} C_VEL
LIN {X 0,Y 304.122,Z 783.762,A -85,B 0,C 180,E1 -16175.785,E2 -16175.785} C_VEL
LIN {X 0,Y 304.153,Z 786.564,A -85,B 0,C 180,E1 -16178.588,E2 -16178.588} C_VEL
LIN {X 0,Y 307.022,Z 800.59,A -85,B 0,C 180,E1 -16179.5,E2 -16179.5} C_VEL
LIN {X 0,Y 309.599,Z 813.662,A -85,B 0,C 180,E1 -16180.612,E2 -16180.612} C_VEL
LIN {X 0,Y 310.347,Z 817.672,A -85,B 0,C 180,E1 -16181.004,E2 -16181.004} C_VEL
LIN {X 0,Y 309.378,Z 830.331,A -85,B 0,C 180,E1 -16182.314,E2 -16182.314} C_VEL
LIN {X 0,Y 308.343,Z 841.781,A -85,B 0,C 180,E1 -16183.81,E2 -16183.81} C_VEL
LIN {X 0,Y 307.227,Z 851.877,A -85,B 0,C 180,E1 -16185.427,E2 -16185.427} C_VEL
LIN {X 0,Y 306.266,Z 860.353,A -85,B 0,C 180,E1 -16187.073,E2 -16187.073} C_VEL
LIN {X 0,Y 305.98,Z 863.252,A -85,B 0,C 180,E1 -16187.718,E2 -16187.718} C_VEL
LIN {X 0,Y 304.946,Z 866.906,A -85,B 0,C 180,E1 -16188.566,E2 -16188.566} C_VEL
LIN {X 0,Y 301.517,Z 872.323,A -85,B 0,C 180,E1 -16189.995,E2 -16189.995} C_VEL
LIN {X 0,Y 298.185,Z 877.209,A -85,B 0,C 180,E1 -16191.529,E2 -16191.529} C_VEL
LIN {X 0,Y 297.319,Z 879.914,A -85,B 0,C 180,E1 -16192.525,E2 -16192.525} C_VEL
LIN {X 0,Y 296.999,Z 884.519,A -85,B 0,C 180,E1 -16194.57,E2 -16194.57} C_VEL
LIN {X 0,Y 296.903,Z 886.959,A -85,B 0,C 180,E1 -16195.929,E2 -16195.929} C_VEL
LIN {X 0,Y 296.804,Z 888.951,A -85,B 0,C 180,E1 -16197.287,E2 -16197.287} C_VEL
LIN {X 0,Y 296.776,Z 890.472,A -85,B 0,C 180,E1 -16198.644,E2 -16198.644} C_VEL
LIN {X 0,Y 296.929,Z 892.327,A -85,B 0,C 180,E1 -16201.358,E2 -16201.358} C_VEL
LIN {X 0,Y 297.118,Z 892.608,A -85,B 0,C 180,E1 -16202.713,E2 -16202.713} C_VEL
LIN {X 0,Y 297.308,Z 892.493,A -85,B 0,C 180,E1 -16204.068,E2 -16204.068} C_VEL
LIN {X 0,Y 297.73,Z 891.122,A -85,B 0,C 180,E1 -16206.78,E2 -16206.78} C_VEL
LIN {X 0,Y 298.752,Z 888.878,A -85,B 0,C 180,E1 -16208.872,E2 -16208.872} C_VEL
LIN {X 0,Y 300.046,Z 884.637,A -85,B 0,C 180,E1 -16211.485,E2 -16211.485} C_VEL
LIN {X 0,Y 301.401,Z 880.215,A -85,B 0,C 180,E1 -16213.486,E2 -16213.486} C_VEL
LIN {X 0,Y 303.489,Z 873.598,A -85,B 0,C 180,E1 -16215.79,E2 -16215.79} C_VEL
LIN {X 0,Y 305.915,Z 865.195,A -85,B 0,C 180,E1 -16218.069,E2 -16218.069} C_VEL
LIN {X 0,Y 308.512,Z 856.251,A -85,B 0,C 180,E1 -16219.982,E2 -16219.982} C_VEL
LIN {X 0,Y 311.201,Z 845.802,A -85,B 0,C 180,E1 -16221.792,E2 -16221.792} C_VEL
LIN {X 0,Y 314.153,Z 833.517,A -85,B 0,C 180,E1 -16223.476,E2 -16223.476} C_VEL
LIN {X 0,Y 314.013,Z 829.98,A -85,B 0,C 180,E1 -16224.047,E2 -16224.047} C_VEL
LIN {X 0,Y 311.535,Z 819.829,A -85,B 0,C 180,E1 -16225.963,E2 -16225.963} C_VEL
LIN {X 0,Y 308.303,Z 811.414,A -85,B 0,C 180,E1 -16227.732,E2 -16227.732} C_VEL
LIN {X 0,Y 304.566,Z 803.81,A -85,B 0,C 180,E1 -16229.56,E2 -16229.56} C_VEL
LIN {X 0,Y 301.926,Z 799.379,A -85,B 0,C 180,E1 -16230.805,E2 -16230.805} C_VEL
LIN {X 0,Y 300.402,Z 796.58,A -85,B 0,C 180,E1 -16231.603,E2 -16231.603} C_VEL
LIN {X 0,Y 300.15,Z 795.714,A -85,B 0,C 180,E1 -16231.793,E2 -16231.793} C_VEL
LIN {X 0,Y 300.36,Z 794.247,A -85,B 0,C 180,E1 -16235.02,E2 -16235.02} C_VEL
LIN {X 0,Y 300.409,Z 793.411,A -85,B 0,C 180,E1 -16237.465,E2 -16237.465} C_VEL
LIN {X 0,Y 300.433,Z 792.792,A -85,B 0,C 180,E1 -16240.921,E2 -16240.921} C_VEL
LIN {X 0,Y 300.508,Z 792.953,A -85,B 0,C 180,E1 -16244.558,E2 -16244.558} C_VEL
LIN {X 0,Y 300.526,Z 793.84,A -85,B 0,C 180,E1 -16247.298,E2 -16247.298} C_VEL
LIN {X 0,Y 300.527,Z 795.869,A -85,B 0,C 180,E1 -16250.511,E2 -16250.511} C_VEL
LIN {X 0,Y 300.767,Z 797.353,A -85,B 0,C 180,E1 -16252.165,E2 -16252.165} C_VEL
LIN {X 0,Y 300.764,Z 800.523,A -85,B 0,C 180,E1 -16254.255,E2 -16254.255} C_VEL
LIN {X 0,Y 299.938,Z 805.909,A -85,B 0,C 180,E1 -16257.517,E2 -16257.517} C_VEL
LIN {X 0,Y 299.907,Z 807.253,A -85,B 0,C 180,E1 -16258.013,E2 -16258.013} C_VEL
LIN {X 0,Y 300.864,Z 811.304,A -85,B 0,C 180,E1 -16258.705,E2 -16258.705} C_VEL
LIN {X 0,Y 301.924,Z 813.473,A -85,B 0,C 180,E1 -16259.196,E2 -16259.196} C_VEL
LIN {X 0,Y 302.969,Z 818.053,A -85,B 0,C 180,E1 -16259.922,E2 -16259.922} C_VEL
LIN {X 0,Y 303.761,Z 819.953,A -85,B 0,C 180,E1 -16260.294,E2 -16260.294} C_VEL
LIN {X 0,Y 306.966,Z 834.61,A -85,B 0,C 180,E1 -16262.545,E2 -16262.545} C_VEL
LIN {X 0,Y 308.632,Z 847.202,A -85,B 0,C 180,E1 -16264.364,E2 -16264.364} C_VEL
LIN {X 0,Y 309.041,Z 858.531,A -85,B 0,C 180,E1 -16265.985,E2 -16265.985} C_VEL
LIN {X 0,Y 307.988,Z 871.387,A -85,B 0,C 180,E1 -16267.882,E2 -16267.882} C_VEL
LIN {X 0,Y 307.426,Z 875.538,A -85,B 0,C 180,E1 -16268.545,E2 -16268.545} C_VEL
LIN {X 0,Y 305.079,Z 884.993,A -85,B 0,C 180,E1 -16270.136,E2 -16270.136} C_VEL
LIN {X 0,Y 302.398,Z 895.668,A -85,B 0,C 180,E1 -16272.344,E2 -16272.344} C_VEL
LIN {X 0,Y 300.508,Z 903.583,A -85,B 0,C 180,E1 -16274.398,E2 -16274.398} C_VEL
LIN {X 0,Y 299.034,Z 909.915,A -85,B 0,C 180,E1 -16276.407,E2 -16276.407} C_VEL
LIN {X 0,Y 297.965,Z 915.082,A -85,B 0,C 180,E1 -16278.435,E2 -16278.435} C_VEL
LIN {X 0,Y 297.255,Z 919.165,A -85,B 0,C 180,E1 -16280.474,E2 -16280.474} C_VEL
LIN {X 0,Y 296.955,Z 921.344,A -85,B 0,C 180,E1 -16281.836,E2 -16281.836} C_VEL
LIN {X 0,Y 296.743,Z 924.033,A -85,B 0,C 180,E1 -16284.119,E2 -16284.119} C_VEL
LIN {X 0,Y 296.699,Z 925.307,A -85,B 0,C 180,E1 -16285.925,E2 -16285.925} C_VEL
LIN {X 0,Y 296.966,Z 926.279,A -85,B 0,C 180,E1 -16288.644,E2 -16288.644} C_VEL
LIN {X 0,Y 296.999,Z 927.094,A -85,B 0,C 180,E1 -16290,E2 -16290} C_VEL
LIN {X 0,Y 296.805,Z 927.463,A -85,B 0,C 180,E1 -16291.357,E2 -16291.357} C_VEL
LIN {X 0,Y 296.66,Z 927.377,A -85,B 0,C 180,E1 -16292.716,E2 -16292.716} C_VEL
LIN {X 0,Y 296.663,Z 926.892,A -85,B 0,C 180,E1 -16294.076,E2 -16294.076} C_VEL
LIN {X 0,Y 296.651,Z 925.792,A -85,B 0,C 180,E1 -16295.706,E2 -16295.706} C_VEL
LIN {X 0,Y 296.925,Z 922.964,A -85,B 0,C 180,E1 -16298.165,E2 -16298.165} C_VEL
LIN {X 0,Y 297.674,Z 918.243,A -85,B 0,C 180,E1 -16300.887,E2 -16300.887} C_VEL
LIN {X 0,Y 298.632,Z 913.506,A -85,B 0,C 180,E1 -16302.919,E2 -16302.919} C_VEL
LIN {X 0,Y 300.282,Z 906.575,A -85,B 0,C 180,E1 -16305.266,E2 -16305.266} C_VEL
LIN {X 0,Y 302.356,Z 897.939,A -85,B 0,C 180,E1 -16307.588,E2 -16307.588} C_VEL
LIN {X 0,Y 304.615,Z 888.896,A -85,B 0,C 180,E1 -16309.545,E2 -16309.545} C_VEL
LIN {X 0,Y 307.517,Z 877.99,A -85,B 0,C 180,E1 -16311.449,E2 -16311.449} C_VEL
LIN {X 0,Y 308.688,Z 871.802,A -85,B 0,C 180,E1 -16312.418,E2 -16312.418} C_VEL
LIN {X 0,Y 309.784,Z 860.302,A -85,B 0,C 180,E1 -16314.102,E2 -16314.102} C_VEL
LIN {X 0,Y 309.448,Z 850.244,A -85,B 0,C 180,E1 -16315.564,E2 -16315.564} C_VEL
LIN {X 0,Y 307.756,Z 838.581,A -85,B 0,C 180,E1 -16317.333,E2 -16317.333} C_VEL
LIN {X 0,Y 305.336,Z 828.426,A -85,B 0,C 180,E1 -16318.994,E2 -16318.994} C_VEL
LIN {X 0,Y 304.166,Z 824.299,A -85,B 0,C 180,E1 -16319.702,E2 -16319.702} C_VEL
LIN {X 0,Y 302.903,Z 820.919,A -85,B 0,C 180,E1 -16320.371,E2 -16320.371} C_VEL
LIN {X 0,Y 302.277,Z 818.754,A -85,B 0,C 180,E1 -16320.764,E2 -16320.764} C_VEL
LIN {X 0,Y 300.752,Z 815.049,A -85,B 0,C 180,E1 -16321.546,E2 -16321.546} C_VEL
LIN {X 0,Y 300.472,Z 813.188,A -85,B 0,C 180,E1 -16321.853,E2 -16321.853} C_VEL
LIN {X 0,Y 301.489,Z 809.008,A -85,B 0,C 180,E1 -16325.323,E2 -16325.323} C_VEL
LIN {X 0,Y 301.879,Z 806.574,A -85,B 0,C 180,E1 -16327.668,E2 -16327.668} C_VEL
LIN {X 0,Y 301.832,Z 803.962,A -85,B 0,C 180,E1 -16330.69,E2 -16330.69} C_VEL
LIN {X 0,Y 301.461,Z 801.519,A -85,B 0,C 180,E1 -16334.379,E2 -16334.379} C_VEL
LIN {X 0,Y 301.116,Z 799.704,A -85,B 0,C 180,E1 -16338.321,E2 -16338.321} C_VEL
LIN {X 0,Y 300.905,Z 798.938,A -85,B 0,C 180,E1 -16340.903,E2 -16340.903} C_VEL
LIN {X 0,Y 300.573,Z 798.439,A -85,B 0,C 180,E1 -16344.227,E2 -16344.227} C_VEL
LIN {X 0,Y 300.085,Z 798.496,A -85,B 0,C 180,E1 -16348.233,E2 -16348.233} C_VEL
LIN {X 0,Y 300.862,Z 800.859,A -85,B 0,C 180,E1 -16348.781,E2 -16348.781} C_VEL
LIN {X 0,Y 303.149,Z 804.195,A -85,B 0,C 180,E1 -16349.89,E2 -16349.89} C_VEL
LIN {X 0,Y 306.625,Z 810.382,A -85,B 0,C 180,E1 -16351.579,E2 -16351.579} C_VEL
LIN {X 0,Y 309.692,Z 816.955,A -85,B 0,C 180,E1 -16353.146,E2 -16353.146} C_VEL
LIN {X 0,Y 312.36,Z 824.278,A -85,B 0,C 180,E1 -16354.69,E2 -16354.69} C_VEL
LIN {X 0,Y 314.019,Z 830.904,A -85,B 0,C 180,E1 -16355.975,E2 -16355.975} C_VEL
LIN {X 0,Y 314.396,Z 834.131,A -85,B 0,C 180,E1 -16356.552,E2 -16356.552} C_VEL
LIN {X 0,Y 311.69,Z 845.408,A -85,B 0,C 180,E1 -16358.099,E2 -16358.099} C_VEL
LIN {X 0,Y 309.196,Z 855.007,A -85,B 0,C 180,E1 -16359.717,E2 -16359.717} C_VEL
LIN {X 0,Y 306.496,Z 864.237,A -85,B 0,C 180,E1 -16361.62,E2 -16361.62} C_VEL
LIN {X 0,Y 304.32,Z 871.766,A -85,B 0,C 180,E1 -16363.565,E2 -16363.565} C_VEL
LIN {X 0,Y 302.13,Z 878.847,A -85,B 0,C 180,E1 -16365.861,E2 -16365.861} C_VEL
LIN {X 0,Y 300.546,Z 883.634,A -85,B 0,C 180,E1 -16367.85,E2 -16367.85} C_VEL
LIN {X 0,Y 299.427,Z 887.384,A -85,B 0,C 180,E1 -16369.86,E2 -16369.86} C_VEL
LIN {X 0,Y 298.429,Z 890.157,A -85,B 0,C 180,E1 -16371.876,E2 -16371.876} C_VEL
LIN {X 0,Y 297.751,Z 891.518,A -85,B 0,C 180,E1 -16373.221,E2 -16373.221} C_VEL
LIN {X 0,Y 297.573,Z 892.406,A -85,B 0,C 180,E1 -16374.578,E2 -16374.578} C_VEL
LIN {X 0,Y 297.431,Z 892.907,A -85,B 0,C 180,E1 -16375.934,E2 -16375.934} C_VEL
LIN {X 0,Y 297.168,Z 893.043,A -85,B 0,C 180,E1 -16377.288,E2 -16377.288} C_VEL
LIN {X 0,Y 296.971,Z 892.788,A -85,B 0,C 180,E1 -16378.643,E2 -16378.643} C_VEL
LIN {X 0,Y 296.864,Z 892.095,A -85,B 0,C 180,E1 -16379.999,E2 -16379.999} C_VEL
LIN {X 0,Y 296.814,Z 890.991,A -85,B 0,C 180,E1 -16381.355,E2 -16381.355} C_VEL
LIN {X 0,Y 296.82,Z 889.489,A -85,B 0,C 180,E1 -16382.713,E2 -16382.713} C_VEL
LIN {X 0,Y 296.98,Z 886.409,A -85,B 0,C 180,E1 -16384.75,E2 -16384.75} C_VEL
LIN {X 0,Y 297.221,Z 882.271,A -85,B 0,C 180,E1 -16386.788,E2 -16386.788} C_VEL
LIN {X 0,Y 297.679,Z 875.963,A -85,B 0,C 180,E1 -16389.168,E2 -16389.168} C_VEL
LIN {X 0,Y 298.407,Z 869.104,A -85,B 0,C 180,E1 -16391.202,E2 -16391.202} C_VEL
LIN {X 0,Y 299.3,Z 860.675,A -85,B 0,C 180,E1 -16393.233,E2 -16393.233} C_VEL
LIN {X 0,Y 300.314,Z 852.153,A -85,B 0,C 180,E1 -16394.916,E2 -16394.916} C_VEL
LIN {X 0,Y 301.438,Z 842.311,A -85,B 0,C 180,E1 -16396.518,E2 -16396.518} C_VEL
LIN {X 0,Y 302.554,Z 830.455,A -85,B 0,C 180,E1 -16398.099,E2 -16398.099} C_VEL
LIN {X 0,Y 303.494,Z 819.709,A -85,B 0,C 180,E1 -16399.252,E2 -16399.252} C_VEL
LIN {X 0,Y 301.397,Z 808.62,A -85,B 0,C 180,E1 -16400.323,E2 -16400.323} C_VEL
LIN {X 0,Y 298.601,Z 794.888,A -85,B 0,C 180,E1 -16401.394,E2 -16401.394} C_VEL
LIN {X 0,Y 297.124,Z 787.653,A -85,B 0,C 180,E1 -16401.87,E2 -16401.87} C_VEL
LIN {X 0,Y 297.219,Z 784.766,A -85,B 0,C 180,E1 -16405.189,E2 -16405.189} C_VEL
LIN {X 0,Y 297.348,Z 784.448,A -85,B 0,C 180,E1 -16406.683,E2 -16406.683} C_VEL
LIN {X 0,Y 297.677,Z 784.402,A -85,B 0,C 180,E1 -16409.721,E2 -16409.721} C_VEL
LIN {X 0,Y 298.061,Z 784.355,A -85,B 0,C 180,E1 -16412.84,E2 -16412.84} C_VEL
LIN {X 0,Y 298.377,Z 784.318,A -85,B 0,C 180,E1 -16416.789,E2 -16416.789} C_VEL
LIN {X 0,Y 298.394,Z 784.312,A -85,B 0,C 180,E1 -16419.486,E2 -16419.486} C_VEL
LIN {X 0,Y 298.394,Z 784.314,A -85,B 0,C 180,E1 -16423.102,E2 -16423.102} C_VEL
LIN {X 0,Y 298.397,Z 784.316,A -85,B 0,C 180,E1 -16426.919,E2 -16426.919} C_VEL
LIN {X 0,Y 298.392,Z 784.317,A -85,B 0,C 180,E1 -16431.006,E2 -16431.006} C_VEL
LIN {X 0,Y 298.411,Z 784.31,A -85,B 0,C 180,E1 -16433.929,E2 -16433.929} C_VEL
LIN {X 0,Y 298.381,Z 784.313,A -85,B 0,C 180,E1 -16437.985,E2 -16437.985} C_VEL
LIN {X 0,Y 298.406,Z 784.311,A -85,B 0,C 180,E1 -16441.898,E2 -16441.898} C_VEL
LIN {X 0,Y 298.432,Z 784.31,A -85,B 0,C 180,E1 -16444.919,E2 -16444.919} C_VEL
LIN {X 0,Y 298.405,Z 784.312,A -85,B 0,C 180,E1 -16447.862,E2 -16447.862} C_VEL
LIN {X 0,Y 298.469,Z 784.303,A -85,B 0,C 180,E1 -16450.752,E2 -16450.752} C_VEL
LIN {X 0,Y 298.577,Z 784.29,A -85,B 0,C 180,E1 -16454.994,E2 -16454.994} C_VEL
LIN {X 0,Y 298.574,Z 784.291,A -85,B 0,C 180,E1 -16459.146,E2 -16459.146} C_VEL
LIN {X 0,Y 298.688,Z 784.28,A -85,B 0,C 180,E1 -16461.884,E2 -16461.884} C_VEL
LIN {X 0,Y 298.616,Z 784.284,A -85,B 0,C 180,E1 -16464.598,E2 -16464.598} C_VEL
LIN {X 0,Y 298.893,Z 784.251,A -85,B 0,C 180,E1 -16468.653,E2 -16468.653} C_VEL
LIN {X 0,Y 298.891,Z 784.251,A -85,B 0,C 180,E1 -16471.347,E2 -16471.347} C_VEL
LIN {X 0,Y 298.723,Z 784.272,A -85,B 0,C 180,E1 -16476.756,E2 -16476.756} C_VEL
LIN {X 0,Y 298.615,Z 784.285,A -85,B 0,C 180,E1 -16479.483,E2 -16479.483} C_VEL
LIN {X 0,Y 298.535,Z 784.294,A -85,B 0,C 180,E1 -16483.616,E2 -16483.616} C_VEL
LIN {X 0,Y 298.475,Z 784.307,A -85,B 0,C 180,E1 -16486.413,E2 -16486.413} C_VEL
LIN {X 0,Y 298.451,Z 784.305,A -85,B 0,C 180,E1 -16489.627,E2 -16489.627} C_VEL
LIN {X 0,Y 298.412,Z 784.31,A -85,B 0,C 180,E1 -16493.602,E2 -16493.602} C_VEL
LIN {X 0,Y 298.4,Z 784.316,A -85,B 0,C 180,E1 -16496.583,E2 -16496.583} C_VEL
LIN {X 0,Y 298.386,Z 784.313,A -85,B 0,C 180,E1 -16499.645,E2 -16499.645} C_VEL
LIN {X 0,Y 298.385,Z 784.317,A -85,B 0,C 180,E1 -16502.802,E2 -16502.802} C_VEL
LIN {X 0,Y 298.438,Z 784.311,A -85,B 0,C 180,E1 -16506.808,E2 -16506.808} C_VEL
LIN {X 0,Y 298.382,Z 784.318,A -85,B 0,C 180,E1 -16511.089,E2 -16511.089} C_VEL
LIN {X 0,Y 298.393,Z 784.317,A -85,B 0,C 180,E1 -16513.105,E2 -16513.105} C_VEL
LIN {X 0,Y 298.398,Z 784.314,A -85,B 0,C 180,E1 -16516.922,E2 -16516.922} C_VEL
LIN {X 0,Y 298.39,Z 784.314,A -85,B 0,C 180,E1 -16521.01,E2 -16521.01} C_VEL
LIN {X 0,Y 298.338,Z 784.321,A -85,B 0,C 180,E1 -16523.921,E2 -16523.921} C_VEL
LIN {X 0,Y 298.109,Z 784.35,A -85,B 0,C 180,E1 -16527.166,E2 -16527.166} C_VEL
LIN {X 0,Y 297.7,Z 784.399,A -85,B 0,C 180,E1 -16530.867,E2 -16530.867} C_VEL
LIN {X 0,Y 297.189,Z 784.463,A -85,B 0,C 180,E1 -16534.809,E2 -16534.809} C_VEL
LIN {X 0,Y 297.053,Z 784.558,A -85,B 0,C 180,E1 -16535.915,E2 -16535.915} C_VEL
LIN {X 0,Y 297.098,Z 786.94,A -85,B 0,C 180,E1 -16538.31,E2 -16538.31} C_VEL
LIN {X 0,Y 299.958,Z 801.024,A -85,B 0,C 180,E1 -16539.247,E2 -16539.247} C_VEL
LIN {X 0,Y 302.545,Z 814.373,A -85,B 0,C 180,E1 -16540.406,E2 -16540.406} C_VEL
LIN {X 0,Y 303.377,Z 819.514,A -85,B 0,C 180,E1 -16540.923,E2 -16540.923} C_VEL
LIN {X 0,Y 302.306,Z 831.625,A -85,B 0,C 180,E1 -16542.236,E2 -16542.236} C_VEL
LIN {X 0,Y 301.09,Z 843.817,A -85,B 0,C 180,E1 -16543.909,E2 -16543.909} C_VEL
LIN {X 0,Y 300.084,Z 852.834,A -85,B 0,C 180,E1 -16545.419,E2 -16545.419} C_VEL
LIN {X 0,Y 298.996,Z 862.694,A -85,B 0,C 180,E1 -16547.444,E2 -16547.444} C_VEL
LIN {X 0,Y 298.143,Z 870.728,A -85,B 0,C 180,E1 -16549.475,E2 -16549.475} C_VEL
LIN {X 0,Y 297.588,Z 876.211,A -85,B 0,C 180,E1 -16551.171,E2 -16551.171} C_VEL
LIN {X 0,Y 297.319,Z 879.914,A -85,B 0,C 180,E1 -16552.525,E2 -16552.525} C_VEL
LIN {X 0,Y 296.494,Z 882.441,A -85,B 0,C 180,E1 -16553.543,E2 -16553.543} C_VEL
LIN {X 0,Y 293.403,Z 885.934,A -85,B 0,C 180,E1 -16555.243,E2 -16555.243} C_VEL
LIN {X 0,Y 290.853,Z 888.239,A -85,B 0,C 180,E1 -16556.661,E2 -16556.661} C_VEL
LIN {X 0,Y 289.768,Z 889.752,A -85,B 0,C 180,E1 -16557.779,E2 -16557.779} C_VEL
LIN {X 0,Y 289.68,Z 890.166,A -85,B 0,C 180,E1 -16558.16,E2 -16558.16} C_VEL
LIN {X 0,Y 289.721,Z 891.892,A -85,B 0,C 180,E1 -16560.001,E2 -16560.001} C_VEL
LIN {X 0,Y 289.841,Z 892.695,A -85,B 0,C 180,E1 -16561.391,E2 -16561.391} C_VEL
LIN {X 0,Y 290.041,Z 893.099,A -85,B 0,C 180,E1 -16562.779,E2 -16562.779} C_VEL
LIN {X 0,Y 290.238,Z 893.068,A -85,B 0,C 180,E1 -16564.167,E2 -16564.167} C_VEL
LIN {X 0,Y 290.73,Z 891.863,A -85,B 0,C 180,E1 -16566.944,E2 -16566.944} C_VEL
LIN {X 0,Y 291.803,Z 889.771,A -85,B 0,C 180,E1 -16569.076,E2 -16569.076} C_VEL
LIN {X 0,Y 292.808,Z 886.951,A -85,B 0,C 180,E1 -16571.072,E2 -16571.072} C_VEL
LIN {X 0,Y 294.124,Z 883.072,A -85,B 0,C 180,E1 -16573.122,E2 -16573.122} C_VEL
LIN {X 0,Y 295.835,Z 878.087,A -85,B 0,C 180,E1 -16575.15,E2 -16575.15} C_VEL
LIN {X 0,Y 298.292,Z 870.793,A -85,B 0,C 180,E1 -16577.483,E2 -16577.483} C_VEL
LIN {X 0,Y 300.315,Z 864.438,A -85,B 0,C 180,E1 -16579.126,E2 -16579.126} C_VEL
LIN {X 0,Y 303.092,Z 855.283,A -85,B 0,C 180,E1 -16581.065,E2 -16581.065} C_VEL
LIN {X 0,Y 305.88,Z 845.177,A -85,B 0,C 180,E1 -16582.809,E2 -16582.809} C_VEL
LIN {X 0,Y 308.448,Z 834.57,A -85,B 0,C 180,E1 -16584.3,E2 -16584.3} C_VEL
LIN {X 0,Y 307.157,Z 827.142,A -85,B 0,C 180,E1 -16585.77,E2 -16585.77} C_VEL
LIN {X 0,Y 304.866,Z 819.244,A -85,B 0,C 180,E1 -16587.456,E2 -16587.456} C_VEL
LIN {X 0,Y 301.27,Z 810.652,A -85,B 0,C 180,E1 -16589.569,E2 -16589.569} C_VEL
LIN {X 0,Y 298.224,Z 805.004,A -85,B 0,C 180,E1 -16591.23,E2 -16591.23} C_VEL
LIN {X 0,Y 296.563,Z 801.629,A -85,B 0,C 180,E1 -16592.239,E2 -16592.239} C_VEL
LIN {X 0,Y 294.472,Z 799.165,A -85,B 0,C 180,E1 -16593.35,E2 -16593.35} C_VEL
LIN {X 0,Y 293.591,Z 796.894,A -85,B 0,C 180,E1 -16594.119,E2 -16594.119} C_VEL
LIN {X 0,Y 293.741,Z 795.772,A -85,B 0,C 180,E1 -16597.856,E2 -16597.856} C_VEL
LIN {X 0,Y 293.805,Z 795.437,A -85,B 0,C 180,E1 -16600.231,E2 -16600.231} C_VEL
LIN {X 0,Y 293.973,Z 795.619,A -85,B 0,C 180,E1 -16603.894,E2 -16603.894} C_VEL
LIN {X 0,Y 294.008,Z 796.267,A -85,B 0,C 180,E1 -16606.114,E2 -16606.114} C_VEL
LIN {X 0,Y 294.039,Z 797.163,A -85,B 0,C 180,E1 -16607.991,E2 -16607.991} C_VEL
LIN {X 0,Y 294.376,Z 800.307,A -85,B 0,C 180,E1 -16611.987,E2 -16611.987} C_VEL
LIN {X 0,Y 294.33,Z 801.971,A -85,B 0,C 180,E1 -16613.348,E2 -16613.348} C_VEL
LIN {X 0,Y 293.853,Z 806.197,A -85,B 0,C 180,E1 -16615.907,E2 -16615.907} C_VEL
LIN {X 0,Y 295.911,Z 812.079,A -85,B 0,C 180,E1 -16617.322,E2 -16617.322} C_VEL
LIN {X 0,Y 297.023,Z 816.593,A -85,B 0,C 180,E1 -16618.174,E2 -16618.174} C_VEL
LIN {X 0,Y 297.703,Z 818.246,A -85,B 0,C 180,E1 -16618.563,E2 -16618.563} C_VEL
LIN {X 0,Y 298.516,Z 822.276,A -85,B 0,C 180,E1 -16619.244,E2 -16619.244} C_VEL
LIN {X 0,Y 299.446,Z 825.802,A -85,B 0,C 180,E1 -16619.9,E2 -16619.9} C_VEL
LIN {X 0,Y 301.686,Z 838.001,A -85,B 0,C 180,E1 -16621.924,E2 -16621.924} C_VEL
LIN {X 0,Y 302.826,Z 848.874,A -85,B 0,C 180,E1 -16623.612,E2 -16623.612} C_VEL
LIN {X 0,Y 303.063,Z 858.924,A -85,B 0,C 180,E1 -16625.147,E2 -16625.147} C_VEL
LIN {X 0,Y 301.903,Z 871.207,A -85,B 0,C 180,E1 -16627.05,E2 -16627.05} C_VEL
LIN {X 0,Y 300.962,Z 877.159,A -85,B 0,C 180,E1 -16628.06,E2 -16628.06} C_VEL
LIN {X 0,Y 298.091,Z 887.895,A -85,B 0,C 180,E1 -16630.01,E2 -16630.01} C_VEL
LIN {X 0,Y 295.618,Z 896.739,A -85,B 0,C 180,E1 -16631.997,E2 -16631.997} C_VEL
LIN {X 0,Y 293.431,Z 905.251,A -85,B 0,C 180,E1 -16634.368,E2 -16634.368} C_VEL
LIN {X 0,Y 291.714,Z 912.012,A -85,B 0,C 180,E1 -16636.769,E2 -16636.769} C_VEL
LIN {X 0,Y 290.696,Z 916.631,A -85,B 0,C 180,E1 -16638.848,E2 -16638.848} C_VEL
LIN {X 0,Y 290.045,Z 920.235,A -85,B 0,C 180,E1 -16640.938,E2 -16640.938} C_VEL
LIN {X 0,Y 289.681,Z 922.873,A -85,B 0,C 180,E1 -16643.032,E2 -16643.032} C_VEL
LIN {X 0,Y 289.629,Z 924.105,A -85,B 0,C 180,E1 -16644.43,E2 -16644.43} C_VEL
LIN {X 0,Y 289.612,Z 924.938,A -85,B 0,C 180,E1 -16645.825,E2 -16645.825} C_VEL
LIN {X 0,Y 289.907,Z 925.597,A -85,B 0,C 180,E1 -16648.611,E2 -16648.611} C_VEL
LIN {X 0,Y 289.942,Z 926.465,A -85,B 0,C 180,E1 -16650,E2 -16650} C_VEL
LIN {X 0,Y 289.719,Z 926.898,A -85,B 0,C 180,E1 -16651.39,E2 -16651.39} C_VEL
LIN {X 0,Y 289.582,Z 926.923,A -85,B 0,C 180,E1 -16652.782,E2 -16652.782} C_VEL
LIN {X 0,Y 289.575,Z 926.504,A -85,B 0,C 180,E1 -16654.175,E2 -16654.175} C_VEL
LIN {X 0,Y 289.671,Z 924.453,A -85,B 0,C 180,E1 -16656.968,E2 -16656.968} C_VEL
LIN {X 0,Y 290.033,Z 921.842,A -85,B 0,C 180,E1 -16659.062,E2 -16659.062} C_VEL
LIN {X 0,Y 290.69,Z 918.271,A -85,B 0,C 180,E1 -16661.152,E2 -16661.152} C_VEL
LIN {X 0,Y 291.695,Z 913.712,A -85,B 0,C 180,E1 -16663.232,E2 -16663.232} C_VEL
LIN {X 0,Y 293.447,Z 907.042,A -85,B 0,C 180,E1 -16665.631,E2 -16665.631} C_VEL
LIN {X 0,Y 295.759,Z 898.285,A -85,B 0,C 180,E1 -16668.099,E2 -16668.099} C_VEL
LIN {X 0,Y 298.027,Z 890.012,A -85,B 0,C 180,E1 -16669.995,E2 -16669.995} C_VEL
LIN {X 0,Y 301.041,Z 879.518,A -85,B 0,C 180,E1 -16671.934,E2 -16671.934} C_VEL
LIN {X 0,Y 302.48,Z 872.589,A -85,B 0,C 180,E1 -16673.084,E2 -16673.084} C_VEL
LIN {X 0,Y 303.692,Z 862.724,A -85,B 0,C 180,E1 -16674.617,E2 -16674.617} C_VEL
LIN {X 0,Y 303.696,Z 853.31,A -85,B 0,C 180,E1 -16676.084,E2 -16676.084} C_VEL
LIN {X 0,Y 302.366,Z 841.77,A -85,B 0,C 180,E1 -16677.961,E2 -16677.961} C_VEL
LIN {X 0,Y 300.68,Z 833.529,A -85,B 0,C 180,E1 -16679.396,E2 -16679.396} C_VEL
LIN {X 0,Y 299.474,Z 828.554,A -85,B 0,C 180,E1 -16680.33,E2 -16680.33} C_VEL
LIN {X 0,Y 298.097,Z 823.952,A -85,B 0,C 180,E1 -16681.244,E2 -16681.244} C_VEL
LIN {X 0,Y 296.707,Z 820.025,A -85,B 0,C 180,E1 -16682.134,E2 -16682.134} C_VEL
LIN {X 0,Y 296.091,Z 817.9,A -85,B 0,C 180,E1 -16682.581,E2 -16682.581} C_VEL
LIN {X 0,Y 294.69,Z 814.818,A -85,B 0,C 180,E1 -16683.413,E2 -16683.413} C_VEL
LIN {X 0,Y 294.144,Z 811.876,A -85,B 0,C 180,E1 -16684.055,E2 -16684.055} C_VEL
LIN {X 0,Y 294.748,Z 809.114,A -85,B 0,C 180,E1 -16686.591,E2 -16686.591} C_VEL
LIN {X 0,Y 294.947,Z 807.5,A -85,B 0,C 180,E1 -16688.282,E2 -16688.282} C_VEL
LIN {X 0,Y 294.947,Z 805.796,A -85,B 0,C 180,E1 -16690.314,E2 -16690.314} C_VEL
LIN {X 0,Y 294.604,Z 803.461,A -85,B 0,C 180,E1 -16693.774,E2 -16693.774} C_VEL
LIN {X 0,Y 294.243,Z 801.519,A -85,B 0,C 180,E1 -16697.769,E2 -16697.769} C_VEL
LIN {X 0,Y 293.91,Z 800.403,A -85,B 0,C 180,E1 -16701.557,E2 -16701.557} C_VEL
LIN {X 0,Y 293.602,Z 799.965,A -85,B 0,C 180,E1 -16704.935,E2 -16704.935} C_VEL
LIN {X 0,Y 293.477,Z 800.139,A -85,B 0,C 180,E1 -16706.01,E2 -16706.01} C_VEL
LIN {X 0,Y 294.323,Z 802.37,A -85,B 0,C 180,E1 -16706.694,E2 -16706.694} C_VEL
LIN {X 0,Y 296.38,Z 804.517,A -85,B 0,C 180,E1 -16707.8,E2 -16707.8} C_VEL
LIN {X 0,Y 297.828,Z 807.547,A -85,B 0,C 180,E1 -16708.724,E2 -16708.724} C_VEL
LIN {X 0,Y 301.055,Z 813.007,A -85,B 0,C 180,E1 -16710.487,E2 -16710.487} C_VEL
LIN {X 0,Y 304.528,Z 820.744,A -85,B 0,C 180,E1 -16712.51,E2 -16712.51} C_VEL
LIN {X 0,Y 307.042,Z 828.21,A -85,B 0,C 180,E1 -16714.22,E2 -16714.22} C_VEL
LIN {X 0,Y 308.554,Z 835.778,A -85,B 0,C 180,E1 -16715.795,E2 -16715.795} C_VEL
LIN {X 0,Y 307.656,Z 840.098,A -85,B 0,C 180,E1 -16716.398,E2 -16716.398} C_VEL
LIN {X 0,Y 304.864,Z 850.509,A -85,B 0,C 180,E1 -16717.999,E2 -16717.999} C_VEL
LIN {X 0,Y 301.859,Z 860.52,A -85,B 0,C 180,E1 -16719.914,E2 -16719.914} C_VEL
LIN {X 0,Y 299.153,Z 868.856,A -85,B 0,C 180,E1 -16721.862,E2 -16721.862} C_VEL
LIN {X 0,Y 296.67,Z 876.557,A -85,B 0,C 180,E1 -16724.19,E2 -16724.19} C_VEL
LIN {X 0,Y 294.829,Z 881.913,A -85,B 0,C 180,E1 -16726.208,E2 -16726.208} C_VEL
LIN {X 0,Y 293.278,Z 886.164,A -85,B 0,C 180,E1 -16728.246,E2 -16728.246} C_VEL
LIN {X 0,Y 292,Z 889.884,A -85,B 0,C 180,E1 -16730.685,E2 -16730.685} C_VEL
LIN {X 0,Y 290.75,Z 892.285,A -85,B 0,C 180,E1 -16733.057,E2 -16733.057} C_VEL
LIN {X 0,Y 290.364,Z 893.5,A -85,B 0,C 180,E1 -16735.835,E2 -16735.835} C_VEL
LIN {X 0,Y 290.094,Z 893.556,A -85,B 0,C 180,E1 -16737.221,E2 -16737.221} C_VEL
LIN {X 0,Y 289.885,Z 893.187,A -85,B 0,C 180,E1 -16738.609,E2 -16738.609} C_VEL
LIN {X 0,Y 289.771,Z 892.403,A -85,B 0,C 180,E1 -16739.999,E2 -16739.999} C_VEL
LIN {X 0,Y 289.722,Z 891.226,A -85,B 0,C 180,E1 -16741.389,E2 -16741.389} C_VEL
LIN {X 0,Y 289.782,Z 888.66,A -85,B 0,C 180,E1 -16743.475,E2 -16743.475} C_VEL
LIN {X 0,Y 289.948,Z 885.097,A -85,B 0,C 180,E1 -16745.562,E2 -16745.562} C_VEL
LIN {X 0,Y 290.262,Z 880.444,A -85,B 0,C 180,E1 -16747.651,E2 -16747.651} C_VEL
LIN {X 0,Y 290.901,Z 873.476,A -85,B 0,C 180,E1 -16750.086,E2 -16750.086} C_VEL
